	__SYSTEM.TYPE_CLASS.TYPE_STRING:
	
	convertResult := TryConvert_LINT_TO_STRING(in, _STRING);
	IF convertResult THEN
		convertAddress := ADR(_STRING);
	END_IF
	
END_CASE

IF convertResult THEN
	memcpy(out.pValue,convertAddress,DINT_TO_UDINT(out.diSize));
END_IF

TryConvert_LINT_TO_Destination := convertResult;

END_FUNCTION

// mobject-converters/Converters/LINT_TO_/TryConvert_LINT_TO_WORD
FUNCTION TryConvert_LINT_TO_WORD : BOOL
VAR_INPUT
	in : LINT;
	out : REFERENCE TO WORD;
END_VAR

IF in > DatatypeLimits.MAX_VALUE_OF_LINT_WHICH_CAN_BE_HELD_IN_A_WORD THEN
	RETURN;
END_IF

IF in < DatatypeLimits.MIN_VALUE_OF_LINT_WHICH_CAN_BE_HELD_IN_A_WORD THEN
	RETURN;
END_IF

out := LINT_TO_WORD(in);
TryConvert_LINT_TO_WORD := TRUE;

END_FUNCTION

// mobject-converters/Converters/LINT_TO_/TryConvert_LINT_TO_DWORD
FUNCTION TryConvert_LINT_TO_DWORD : BOOL
VAR_INPUT
	in : LINT;
	out : REFERENCE TO DWORD;
END_VAR

IF in > DatatypeLimits.MAX_VALUE_OF_LINT_WHICH_CAN_BE_HELD_IN_A_DWORD THEN
	RETURN;
END_IF

IF in < DatatypeLimits.MIN_VALUE_OF_LINT_WHICH_CAN_BE_HELD_IN_A_DWORD THEN
	RETURN;
END_IF

out := LINT_TO_DWORD(in);
TryConvert_LINT_TO_DWORD := TRUE;

END_FUNCTION

// mobject-converters/Converters/LINT_TO_/TryConvert_LINT_TO_LWORD
FUNCTION TryConvert_LINT_TO_LWORD : BOOL
VAR_INPUT
	in : LINT;
	out : REFERENCE TO LWORD;
END_VAR

IF in < DatatypeLimits.MIN_VALUE_OF_LINT_WHICH_CAN_BE_HELD_IN_A_LWORD THEN
	RETURN;
END_IF

out := LINT_TO_LWORD(in);
TryConvert_LINT_TO_LWORD := TRUE;

END_FUNCTION

// mobject-converters/Converters/LINT_TO_/TryConvert_LINT_TO_SINT
FUNCTION TryConvert_LINT_TO_SINT : BOOL
VAR_INPUT
	in : LINT;
	out : REFERENCE TO SINT;
END_VAR

IF in > DatatypeLimits.MAX_VALUE_OF_LINT_WHICH_CAN_BE_HELD_IN_A_SINT THEN
	RETURN;
END_IF

IF in < DatatypeLimits.MIN_VALUE_OF_LINT_WHICH_CAN_BE_HELD_IN_A_SINT THEN
	RETURN;
END_IF

out := LINT_TO_SINT(in);
TryConvert_LINT_TO_SINT := TRUE;

END_FUNCTION

// mobject-converters/Converters/LINT_TO_/TryConvert_LINT_TO_INT
FUNCTION TryConvert_LINT_TO_INT : BOOL
VAR_INPUT
	in : LINT;
	out : REFERENCE TO INT;
END_VAR

IF in > DatatypeLimits.MAX_VALUE_OF_LINT_WHICH_CAN_BE_HELD_IN_A_INT THEN
	RETURN;
END_IF

IF in < DatatypeLimits.MIN_VALUE_OF_LINT_WHICH_CAN_BE_HELD_IN_A_INT THEN
	RETURN;
END_IF

out := LINT_TO_INT(in);
TryConvert_LINT_TO_INT := TRUE;

END_FUNCTION

// mobject-converters/Converters/LINT_TO_/TryConvert_LINT_TO_DINT
FUNCTION TryConvert_LINT_TO_DINT : BOOL
VAR_INPUT
	in : LINT;
	out : REFERENCE TO DINT;
END_VAR

IF in > DatatypeLimits.MAX_VALUE_OF_LINT_WHICH_CAN_BE_HELD_IN_A_DINT THEN
	RETURN;
END_IF

IF in < DatatypeLimits.MIN_VALUE_OF_LINT_WHICH_CAN_BE_HELD_IN_A_DINT THEN
	RETURN;
END_IF

out := LINT_TO_DINT(in);
TryConvert_LINT_TO_DINT := TRUE;

END_FUNCTION

// mobject-converters/Converters/LINT_TO_/TryConvert_LINT_TO_LINT
FUNCTION TryConvert_LINT_TO_LINT : BOOL
VAR_INPUT
	in : LINT;
	out : REFERENCE TO LINT;
END_VAR

out := in;
TryConvert_LINT_TO_LINT := TRUE;

END_FUNCTION

// mobject-converters/Converters/LINT_TO_/TryConvert_LINT_TO_USINT
FUNCTION TryConvert_LINT_TO_USINT : BOOL
VAR_INPUT
	in : LINT;
	out : REFERENCE TO USINT;
END_VAR

IF in > DatatypeLimits.MAX_VALUE_OF_LINT_WHICH_CAN_BE_HELD_IN_A_USINT THEN
	RETURN;
END_IF

IF in < DatatypeLimits.MIN_VALUE_OF_LINT_WHICH_CAN_BE_HELD_IN_A_USINT THEN
	RETURN;
END_IF

out := LINT_TO_USINT(in);
TryConvert_LINT_TO_USINT := TRUE;

END_FUNCTION

// mobject-converters/Converters/LINT_TO_/TryConvert_LINT_TO_UINT
FUNCTION TryConvert_LINT_TO_UINT : BOOL
VAR_INPUT
	in : LINT;
	out : REFERENCE TO UINT;
END_VAR

IF in > DatatypeLimits.MAX_VALUE_OF_LINT_WHICH_CAN_BE_HELD_IN_A_UINT THEN
	RETURN;
END_IF

IF in < DatatypeLimits.MIN_VALUE_OF_LINT_WHICH_CAN_BE_HELD_IN_A_UINT THEN
	RETURN;
END_IF

out := LINT_TO_UINT(in);
TryConvert_LINT_TO_UINT := TRUE;

END_FUNCTION

// mobject-converters/Converters/LINT_TO_/TryConvert_LINT_TO_UDINT
FUNCTION TryConvert_LINT_TO_UDINT : BOOL
VAR_INPUT
	in : LINT;
	out : REFERENCE TO UDINT;
END_VAR

IF in > DatatypeLimits.MAX_VALUE_OF_LINT_WHICH_CAN_BE_HELD_IN_A_UDINT THEN
	RETURN;
END_IF

IF in < DatatypeLimits.MIN_VALUE_OF_LINT_WHICH_CAN_BE_HELD_IN_A_UDINT THEN
	RETURN;
END_IF

out := LINT_TO_UDINT(in);
TryConvert_LINT_TO_UDINT := TRUE;

END_FUNCTION

// mobject-converters/Converters/LINT_TO_/TryConvert_LINT_TO_ULINT
FUNCTION TryConvert_LINT_TO_ULINT : BOOL
VAR_INPUT
	in : LINT;
	out : REFERENCE TO ULINT;
END_VAR

IF in < DatatypeLimits.MIN_VALUE_OF_LINT_WHICH_CAN_BE_HELD_IN_A_ULINT THEN
	RETURN;
END_IF

out := LINT_TO_ULINT(in);
TryConvert_LINT_TO_ULINT := TRUE;

END_FUNCTION

// mobject-converters/Converters/LINT_TO_/TryConvert_LINT_TO_REAL
FUNCTION TryConvert_LINT_TO_REAL : BOOL
VAR_INPUT
	in : LINT;
	out : REFERENCE TO REAL;
END_VAR

out := LINT_TO_REAL(in);
TryConvert_LINT_TO_REAL := TRUE;

END_FUNCTION

// mobject-converters/Converters/LINT_TO_/TryConvert_LINT_TO_LREAL
FUNCTION TryConvert_LINT_TO_LREAL : BOOL
VAR_INPUT
	in : LINT;
	out : REFERENCE TO LREAL;
END_VAR

out := LINT_TO_LREAL(in);
TryConvert_LINT_TO_LREAL := TRUE;

END_FUNCTION

// mobject-converters/Converters/LINT_TO_/TryConvert_LINT_TO_TIME
FUNCTION TryConvert_LINT_TO_TIME : BOOL
VAR_INPUT
	in : LINT;
	out : REFERENCE TO TIME;
END_VAR

IF in > DatatypeLimits.MAX_VALUE_OF_LINT_WHICH_CAN_BE_HELD_IN_A_TIME THEN
	RETURN;
END_IF

IF in < DatatypeLimits.MIN_VALUE_OF_LINT_WHICH_CAN_BE_HELD_IN_A_TIME THEN
	RETURN;
END_IF

out := LINT_TO_TIME(in);
TryConvert_LINT_TO_TIME := TRUE;

END_FUNCTION

// mobject-converters/Converters/LINT_TO_/TryConvert_LINT_TO_TOD
FUNCTION TryConvert_LINT_TO_TOD : BOOL
VAR_INPUT
	in : LINT;
	out : REFERENCE TO TOD;
END_VAR

IF in > DatatypeLimits.MAX_VALUE_OF_LINT_WHICH_CAN_BE_HELD_IN_A_TOD THEN
	RETURN;
END_IF

IF in < DatatypeLimits.MIN_VALUE_OF_LINT_WHICH_CAN_BE_HELD_IN_A_TOD THEN
	RETURN;
END_IF

out := LINT_TO_TOD(in);
TryConvert_LINT_TO_TOD := TRUE;

END_FUNCTION

// mobject-converters/Converters/LINT_TO_/TryConvert_LINT_TO_DT
FUNCTION TryConvert_LINT_TO_DT : BOOL
VAR_INPUT
	in : LINT;
	out : REFERENCE TO DT;
END_VAR

IF in > DatatypeLimits.MAX_VALUE_OF_LINT_WHICH_CAN_BE_HELD_IN_A_DT THEN
	RETURN;
END_IF

IF in < DatatypeLimits.MIN_VALUE_OF_LINT_WHICH_CAN_BE_HELD_IN_A_DT THEN
	RETURN;
END_IF

out := LINT_TO_DT(in);
TryConvert_LINT_TO_DT := TRUE;

END_FUNCTION

// mobject-converters/Converters/LINT_TO_/TryConvert_LINT_TO_STRING
FUNCTION TryConvert_LINT_TO_STRING : BOOL
VAR_INPUT
	in : LINT;
	out : REFERENCE TO STRING;
END_VAR

out := LINT_TO_STRING(in);
TryConvert_LINT_TO_STRING := TRUE;

END_FUNCTION

// mobject-converters/Converters/LREAL_TO_/TryConvert_LREAL_TO_BOOL
FUNCTION TryConvert_LREAL_TO_BOOL : BOOL
VAR_INPUT
	in : LREAL;
	out : REFERENCE TO BOOL;
END_VAR

out := LREAL_TO_BOOL(in);
TryConvert_LREAL_TO_BOOL := TRUE;

END_FUNCTION

// mobject-converters/Converters/LREAL_TO_/TryConvert_LREAL_TO_BYTE
FUNCTION TryConvert_LREAL_TO_BYTE : BOOL
VAR_INPUT
	in : LREAL;
	out : REFERENCE TO BYTE;
END_VAR

IF in > DatatypeLimits.MAX_VALUE_OF_LREAL_WHICH_CAN_BE_HELD_IN_A_BYTE THEN
	RETURN;
END_IF

IF in < DatatypeLimits.MIN_VALUE_OF_LREAL_WHICH_CAN_BE_HELD_IN_A_BYTE THEN
	RETURN;
END_IF

out := LREAL_TO_BYTE(in);
TryConvert_LREAL_TO_BYTE := TRUE;

END_FUNCTION

// mobject-converters/Converters/LREAL_TO_/TryConvert_LREAL_TO_DATE
FUNCTION TryConvert_LREAL_TO_DATE : BOOL
VAR_INPUT
	in : LREAL;
	out : REFERENCE TO DATE;
END_VAR

IF in > DatatypeLimits.MAX_VALUE_OF_LREAL_WHICH_CAN_BE_HELD_IN_A_DATE THEN
	RETURN;
END_IF

IF in < DatatypeLimits.MIN_VALUE_OF_LREAL_WHICH_CAN_BE_HELD_IN_A_DATE THEN
	RETURN;
END_IF

out := LREAL_TO_DATE(in);
TryConvert_LREAL_TO_DATE := TRUE;

END_FUNCTION

// mobject-converters/Converters/LREAL_TO_/TryConvert_LREAL_TO_Destination
FUNCTION TryConvert_LREAL_TO_Destination : BOOL
VAR_INPUT
	in : LREAL;
	out : ANY;
END_VAR
VAR
	convertResult : BOOL := FALSE;
	convertAddress : PVOID;
	_BOOL : BOOL;
	_BYTE : BYTE;
	_WORD : WORD;
	_DWORD : DWORD;
	_LWORD : LWORD;
	_SINT : SINT;
	_INT : INT;
	_DINT : DINT;
	_LINT : LINT;
	_USINT : USINT;
	_UINT : UINT;
	_UDINT : UDINT;
	_ULINT : ULINT;
	_REAL : REAL;
	_LREAL : LREAL;
	_TIME : TIME;
	_TOD : TOD;
	_DATE : DATE;
	_DT : DT;
	_STRING : STRING;
END_VAR

CASE out.TypeClass OF
	__SYSTEM.TYPE_CLASS.TYPE_BOOL:
	
	convertResult := TryConvert_LREAL_TO_BOOL(in, _BOOL);
	IF convertResult THEN
		convertAddress := ADR(_BOOL);
	END_IF
	
	__SYSTEM.TYPE_CLASS.TYPE_BYTE:
	
	convertResult := TryConvert_LREAL_TO_BYTE(in, _BYTE);
	IF convertResult THEN
		convertAddress := ADR(_BYTE);
	END_IF
	
	__SYSTEM.TYPE_CLASS.TYPE_WORD:
	
	convertResult := TryConvert_LREAL_TO_WORD(in, _WORD);
	IF convertResult THEN
		convertAddress := ADR(_WORD);
	END_IF
	
	__SYSTEM.TYPE_CLASS.TYPE_DWORD:
	
	convertResult := TryConvert_LREAL_TO_DWORD(in, _DWORD);
	IF convertResult THEN
		convertAddress := ADR(_DWORD);
	END_IF
	
	__SYSTEM.TYPE_CLASS.TYPE_LWORD:
	
	convertResult := TryConvert_LREAL_TO_LWORD(in, _LWORD);
	IF convertResult THEN
		convertAddress := ADR(_LWORD);
	END_IF
	
	__SYSTEM.TYPE_CLASS.TYPE_SINT:
	
	convertResult := TryConvert_LREAL_TO_SINT(in, _SINT);
	IF convertResult THEN
		convertAddress := ADR(_SINT);
	END_IF
	
	__SYSTEM.TYPE_CLASS.TYPE_INT:
	
	convertResult := TryConvert_LREAL_TO_INT(in, _INT);
	IF convertResult THEN
		convertAddress := ADR(_INT);
	END_IF
	
	__SYSTEM.TYPE_CLASS.TYPE_DINT:
	
	convertResult := TryConvert_LREAL_TO_DINT(in, _DINT);
	IF convertResult THEN
		convertAddress := ADR(_DINT);
	END_IF
	
	__SYSTEM.TYPE_CLASS.TYPE_LINT:
	
	convertResult := TryConvert_LREAL_TO_LINT(in, _LINT);
	IF convertResult THEN
		convertAddress := ADR(_LINT);
	END_IF
	
	__SYSTEM.TYPE_CLASS.TYPE_USINT:
	
	convertResult := TryConvert_LREAL_TO_USINT(in, _USINT);
	IF convertResult THEN
		convertAddress := ADR(_USINT);
	END_IF
	
	__SYSTEM.TYPE_CLASS.TYPE_UINT:
	
	convertResult := TryConvert_LREAL_TO_UINT(in, _UINT);
	IF convertResult THEN
		convertAddress := ADR(_UINT);
	END_IF
	
	__SYSTEM.TYPE_CLASS.TYPE_UDINT:
	
	convertResult := TryConvert_LREAL_TO_UDINT(in, _UDINT);
	IF convertResult THEN
		convertAddress := ADR(_UDINT);
	END_IF
	
	__SYSTEM.TYPE_CLASS.TYPE_ULINT:
	
	convertResult := TryConvert_LREAL_TO_ULINT(in, _ULINT);
	IF convertResult THEN
		convertAddress := ADR(_ULINT);
	END_IF
	
	__SYSTEM.TYPE_CLASS.TYPE_REAL:
	
	convertResult := TryConvert_LREAL_TO_REAL(in, _REAL);
	IF convertResult THEN
		convertAddress := ADR(_REAL);
	END_IF
	
	__SYSTEM.TYPE_CLASS.TYPE_LREAL:
	
	convertResult := TryConvert_LREAL_TO_LREAL(in, _LREAL);
	IF convertResult THEN
		convertAddress := ADR(_LREAL);
	END_IF
	
	__SYSTEM.TYPE_CLASS.TYPE_TIME:
	
	convertResult := TryConvert_LREAL_TO_TIME(in, _TIME);
	IF convertResult THEN
		convertAddress := ADR(_TIME);
	END_IF
	
	__SYSTEM.TYPE_CLASS.TYPE_TIMEOFDAY:
	
	convertResult := TryConvert_LREAL_TO_TOD(in, _TOD);
	IF convertResult THEN
		convertAddress := ADR(_TOD);
	END_IF
	
	__SYSTEM.TYPE_CLASS.TYPE_DATE:
	
	convertResult := TryConvert_LREAL_TO_DATE(in, _DATE);
	IF convertResult THEN
		convertAddress := ADR(_DATE);
	END_IF
	
	__SYSTEM.TYPE_CLASS.TYPE_DATEANDTIME:
	
	convertResult := TryConvert_LREAL_TO_DT(in, _DT);
	IF convertResult THEN
		convertAddress := ADR(_DT);
	END_IF
	
	__SYSTEM.TYPE_CLASS.TYPE_STRING:
	
	convertResult := TryConvert_LREAL_TO_STRING(in, _STRING);
	IF convertResult THEN
		convertAddress := ADR(_STRING);
	END_IF
	
END_CASE

IF convertResult THEN
	memcpy(out.pValue,convertAddress,DINT_TO_UDINT(out.diSize));
END_IF

TryConvert_LREAL_TO_Destination := convertResult;

END_FUNCTION

// mobject-converters/Converters/LREAL_TO_/TryConvert_LREAL_TO_WORD
FUNCTION TryConvert_LREAL_TO_WORD : BOOL
VAR_INPUT
	in : LREAL;
	out : REFERENCE TO WORD;
END_VAR

IF in > DatatypeLimits.MAX_VALUE_OF_LREAL_WHICH_CAN_BE_HELD_IN_A_WORD THEN
	RETURN;
END_IF

IF in < DatatypeLimits.MIN_VALUE_OF_LREAL_WHICH_CAN_BE_HELD_IN_A_WORD THEN
	RETURN;
END_IF

out := LREAL_TO_WORD(in);
TryConvert_LREAL_TO_WORD := TRUE;

END_FUNCTION

// mobject-converters/Converters/LREAL_TO_/TryConvert_LREAL_TO_DWORD
FUNCTION TryConvert_LREAL_TO_DWORD : BOOL
VAR_INPUT
	in : LREAL;
	out : REFERENCE TO DWORD;
END_VAR

IF in > DatatypeLimits.MAX_VALUE_OF_LREAL_WHICH_CAN_BE_HELD_IN_A_DWORD THEN
	RETURN;
END_IF

IF in < DatatypeLimits.MIN_VALUE_OF_LREAL_WHICH_CAN_BE_HELD_IN_A_DWORD THEN
	RETURN;
END_IF

out := LREAL_TO_DWORD(in);
TryConvert_LREAL_TO_DWORD := TRUE;

END_FUNCTION

// mobject-converters/Converters/LREAL_TO_/TryConvert_LREAL_TO_LWORD
FUNCTION TryConvert_LREAL_TO_LWORD : BOOL
VAR_INPUT
	in : LREAL;
	out : REFERENCE TO LWORD;
END_VAR

IF in > DatatypeLimits.MAX_VALUE_OF_LREAL_WHICH_CAN_BE_HELD_IN_A_LWORD THEN
	RETURN;
END_IF

IF in < DatatypeLimits.MIN_VALUE_OF_LREAL_WHICH_CAN_BE_HELD_IN_A_LWORD THEN
	RETURN;
END_IF

out := LREAL_TO_LWORD(in);
TryConvert_LREAL_TO_LWORD := TRUE;

END_FUNCTION

// mobject-converters/Converters/LREAL_TO_/TryConvert_LREAL_TO_SINT
FUNCTION TryConvert_LREAL_TO_SINT : BOOL
VAR_INPUT
	in : LREAL;
	out : REFERENCE TO SINT;
END_VAR

IF in > DatatypeLimits.MAX_VALUE_OF_LREAL_WHICH_CAN_BE_HELD_IN_A_SINT THEN
	RETURN;
END_IF

IF in < DatatypeLimits.MIN_VALUE_OF_LREAL_WHICH_CAN_BE_HELD_IN_A_SINT THEN
	RETURN;
END_IF

out := LREAL_TO_SINT(in);
TryConvert_LREAL_TO_SINT := TRUE;

END_FUNCTION

// mobject-converters/Converters/LREAL_TO_/TryConvert_LREAL_TO_INT
FUNCTION TryConvert_LREAL_TO_INT : BOOL
VAR_INPUT
	in : LREAL;
	out : REFERENCE TO INT;
END_VAR

IF in > DatatypeLimits.MAX_VALUE_OF_LREAL_WHICH_CAN_BE_HELD_IN_A_INT THEN
	RETURN;
END_IF

IF in < DatatypeLimits.MIN_VALUE_OF_LREAL_WHICH_CAN_BE_HELD_IN_A_INT THEN
	RETURN;
END_IF

out := LREAL_TO_INT(in);
TryConvert_LREAL_TO_INT := TRUE;

END_FUNCTION

// mobject-converters/Converters/LREAL_TO_/TryConvert_LREAL_TO_DINT
FUNCTION TryConvert_LREAL_TO_DINT : BOOL
VAR_INPUT
	in : LREAL;
	out : REFERENCE TO DINT;
END_VAR

IF in > DatatypeLimits.MAX_VALUE_OF_LREAL_WHICH_CAN_BE_HELD_IN_A_DINT THEN
	RETURN;
END_IF

IF in < DatatypeLimits.MIN_VALUE_OF_LREAL_WHICH_CAN_BE_HELD_IN_A_DINT THEN
	RETURN;
END_IF

out := LREAL_TO_DINT(in);
TryConvert_LREAL_TO_DINT := TRUE;

END_FUNCTION

// mobject-converters/Converters/LREAL_TO_/TryConvert_LREAL_TO_LINT
FUNCTION TryConvert_LREAL_TO_LINT : BOOL
VAR_INPUT
	in : LREAL;
	out : REFERENCE TO LINT;
END_VAR

IF in > DatatypeLimits.MAX_VALUE_OF_LREAL_WHICH_CAN_BE_HELD_IN_A_LINT THEN
	RETURN;
END_IF

IF in < DatatypeLimits.MIN_VALUE_OF_LREAL_WHICH_CAN_BE_HELD_IN_A_LINT THEN
	RETURN;
END_IF

out := LREAL_TO_LINT(in);
TryConvert_LREAL_TO_LINT := TRUE;

END_FUNCTION

// mobject-converters/Converters/LREAL_TO_/TryConvert_LREAL_TO_USINT
FUNCTION TryConvert_LREAL_TO_USINT : BOOL
VAR_INPUT
	in : LREAL;
	out : REFERENCE TO USINT;
END_VAR

IF in > DatatypeLimits.MAX_VALUE_OF_LREAL_WHICH_CAN_BE_HELD_IN_A_USINT THEN
	RETURN;
END_IF

IF in < DatatypeLimits.MIN_VALUE_OF_LREAL_WHICH_CAN_BE_HELD_IN_A_USINT THEN
	RETURN;
END_IF

out := LREAL_TO_USINT(in);
TryConvert_LREAL_TO_USINT := TRUE;

END_FUNCTION

// mobject-converters/Converters/LREAL_TO_/TryConvert_LREAL_TO_UINT
FUNCTION TryConvert_LREAL_TO_UINT : BOOL
VAR_INPUT
	in : LREAL;
	out : REFERENCE TO UINT;
END_VAR

IF in > DatatypeLimits.MAX_VALUE_OF_LREAL_WHICH_CAN_BE_HELD_IN_A_UINT THEN
	RETURN;
END_IF

IF in < DatatypeLimits.MIN_VALUE_OF_LREAL_WHICH_CAN_BE_HELD_IN_A_UINT THEN
	RETURN;
END_IF

out := LREAL_TO_UINT(in);
TryConvert_LREAL_TO_UINT := TRUE;

END_FUNCTION

// mobject-converters/Converters/LREAL_TO_/TryConvert_LREAL_TO_UDINT
FUNCTION TryConvert_LREAL_TO_UDINT : BOOL
VAR_INPUT
	in : LREAL;
	out : REFERENCE TO UDINT;
END_VAR

IF in > DatatypeLimits.MAX_VALUE_OF_LREAL_WHICH_CAN_BE_HELD_IN_A_UDINT THEN
	RETURN;
END_IF

IF in < DatatypeLimits.MIN_VALUE_OF_LREAL_WHICH_CAN_BE_HELD_IN_A_UDINT THEN
	RETURN;
END_IF

out := LREAL_TO_UDINT(in);
TryConvert_LREAL_TO_UDINT := TRUE;

END_FUNCTION

// mobject-converters/Converters/LREAL_TO_/TryConvert_LREAL_TO_ULINT
FUNCTION TryConvert_LREAL_TO_ULINT : BOOL
VAR_INPUT
	in : LREAL;
	out : REFERENCE TO ULINT;
END_VAR

IF in > DatatypeLimits.MAX_VALUE_OF_LREAL_WHICH_CAN_BE_HELD_IN_A_ULINT THEN
	RETURN;
END_IF

IF in < DatatypeLimits.MIN_VALUE_OF_LREAL_WHICH_CAN_BE_HELD_IN_A_ULINT THEN
	RETURN;
END_IF

out := LREAL_TO_ULINT(in);
TryConvert_LREAL_TO_ULINT := TRUE;

END_FUNCTION

// mobject-converters/Converters/LREAL_TO_/TryConvert_LREAL_TO_REAL
FUNCTION TryConvert_LREAL_TO_REAL : BOOL
VAR_INPUT
	in : LREAL;
	out : REFERENCE TO REAL;
END_VAR

IF in > DatatypeLimits.MAX_VALUE_OF_LREAL_WHICH_CAN_BE_HELD_IN_A_REAL THEN
	RETURN;
END_IF

IF in < DatatypeLimits.MIN_VALUE_OF_LREAL_WHICH_CAN_BE_HELD_IN_A_REAL THEN
	RETURN;
END_IF

out := LREAL_TO_REAL(in);
TryConvert_LREAL_TO_REAL := TRUE;

END_FUNCTION

// mobject-converters/Converters/LREAL_TO_/TryConvert_LREAL_TO_LREAL
FUNCTION TryConvert_LREAL_TO_LREAL : BOOL
VAR_INPUT
	in : LREAL;
	out : REFERENCE TO LREAL;
END_VAR

out := in;
TryConvert_LREAL_TO_LREAL := TRUE;

END_FUNCTION

// mobject-converters/Converters/LREAL_TO_/TryConvert_LREAL_TO_TIME
FUNCTION TryConvert_LREAL_TO_TIME : BOOL
VAR_INPUT
	in : LREAL;
	out : REFERENCE TO TIME;
END_VAR

IF in > DatatypeLimits.MAX_VALUE_OF_LREAL_WHICH_CAN_BE_HELD_IN_A_TIME THEN
	RETURN;
END_IF

IF in < DatatypeLimits.MIN_VALUE_OF_LREAL_WHICH_CAN_BE_HELD_IN_A_TIME THEN
	RETURN;
END_IF

out := LREAL_TO_TIME(in);
TryConvert_LREAL_TO_TIME := TRUE;

END_FUNCTION

// mobject-converters/Converters/LREAL_TO_/TryConvert_LREAL_TO_TOD
FUNCTION TryConvert_LREAL_TO_TOD : BOOL
VAR_INPUT
	in : LREAL;
	out : REFERENCE TO TOD;
END_VAR

IF in > DatatypeLimits.MAX_VALUE_OF_LREAL_WHICH_CAN_BE_HELD_IN_A_TOD THEN
	RETURN;
END_IF

IF in < DatatypeLimits.MIN_VALUE_OF_LREAL_WHICH_CAN_BE_HELD_IN_A_TOD THEN
	RETURN;
END_IF

out := LREAL_TO_TOD(in);
TryConvert_LREAL_TO_TOD := TRUE;

END_FUNCTION

// mobject-converters/Converters/LREAL_TO_/TryConvert_LREAL_TO_DT
FUNCTION TryConvert_LREAL_TO_DT : BOOL
VAR_INPUT
	in : LREAL;
	out : REFERENCE TO DT;
END_VAR

IF in > DatatypeLimits.MAX_VALUE_OF_LREAL_WHICH_CAN_BE_HELD_IN_A_DT THEN
	RETURN;
END_IF

IF in < DatatypeLimits.MIN_VALUE_OF_LREAL_WHICH_CAN_BE_HELD_IN_A_DT THEN
	RETURN;
END_IF

out := LREAL_TO_DT(in);
TryConvert_LREAL_TO_DT := TRUE;

END_FUNCTION

// mobject-converters/Converters/LREAL_TO_/TryConvert_LREAL_TO_STRING
FUNCTION TryConvert_LREAL_TO_STRING : BOOL
VAR_INPUT
	in : LREAL;
	out : REFERENCE TO STRING;
END_VAR

IF in > DatatypeLimits.MAX_VALUE_OF_LREAL_WHICH_CAN_BE_HELD_IN_A_STRING THEN
	RETURN;
END_IF

IF in < DatatypeLimits.MIN_VALUE_OF_LREAL_WHICH_CAN_BE_HELD_IN_A_STRING THEN
	RETURN;
END_IF

out := LREAL_TO_STRING(in);
TryConvert_LREAL_TO_STRING := TRUE;

END_FUNCTION

// mobject-converters/Converters/LWORD_TO_/TryConvert_LWORD_TO_BOOL
FUNCTION TryConvert_LWORD_TO_BOOL : BOOL
VAR_INPUT
	in : LWORD;
	out : REFERENCE TO BOOL;
END_VAR

out := LWORD_TO_BOOL(in);
TryConvert_LWORD_TO_BOOL := TRUE;

END_FUNCTION

// mobject-converters/Converters/LWORD_TO_/TryConvert_LWORD_TO_BYTE
FUNCTION TryConvert_LWORD_TO_BYTE : BOOL
VAR_INPUT
	in : LWORD;
	out : REFERENCE TO BYTE;
END_VAR

IF in > DatatypeLimits.MAX_VALUE_OF_LWORD_WHICH_CAN_BE_HELD_IN_A_BYTE THEN
	RETURN;
END_IF

out := LWORD_TO_BYTE(in);
TryConvert_LWORD_TO_BYTE := TRUE;

END_FUNCTION

// mobject-converters/Converters/LWORD_TO_/TryConvert_LWORD_TO_DATE
FUNCTION TryConvert_LWORD_TO_DATE : BOOL
VAR_INPUT
	in : LWORD;
	out : REFERENCE TO DATE;
END_VAR

IF in > DatatypeLimits.MAX_VALUE_OF_LWORD_WHICH_CAN_BE_HELD_IN_A_DATE THEN
	RETURN;
END_IF

out := LWORD_TO_DATE(in);
TryConvert_LWORD_TO_DATE := TRUE;

END_FUNCTION

// mobject-converters/Converters/LWORD_TO_/TryConvert_LWORD_TO_Destination
FUNCTION TryConvert_LWORD_TO_Destination : BOOL
VAR_INPUT
	in : LWORD;
	out : ANY;
END_VAR
VAR
	convertResult : BOOL := FALSE;
	convertAddress : PVOID;
	_BOOL : BOOL;
	_BYTE : BYTE;
	_WORD : WORD;
	_DWORD : DWORD;
	_LWORD : LWORD;
	_SINT : SINT;
	_INT : INT;
	_DINT : DINT;
	_LINT : LINT;
	_USINT : USINT;
	_UINT : UINT;
	_UDINT : UDINT;
	_ULINT : ULINT;
	_REAL : REAL;
	_LREAL : LREAL;
	_TIME : TIME;
	_TOD : TOD;
	_DATE : DATE;
	_DT : DT;
	_STRING : STRING;
END_VAR

CASE out.TypeClass OF
	__SYSTEM.TYPE_CLASS.TYPE_BOOL:
	
	convertResult := TryConvert_LWORD_TO_BOOL(in, _BOOL);
	IF convertResult THEN
		convertAddress := ADR(_BOOL);
	END_IF
	
	__SYSTEM.TYPE_CLASS.TYPE_BYTE:
	
	convertResult := TryConvert_LWORD_TO_BYTE(in, _BYTE);
	IF convertResult THEN
		convertAddress := ADR(_BYTE);
	END_IF
	
	__SYSTEM.TYPE_CLASS.TYPE_WORD:
	
	convertResult := TryConvert_LWORD_TO_WORD(in, _WORD);
	IF convertResult THEN
		convertAddress := ADR(_WORD);
	END_IF
	
	__SYSTEM.TYPE_CLASS.TYPE_DWORD:
	
	convertResult := TryConvert_LWORD_TO_DWORD(in, _DWORD);
	IF convertResult THEN
		convertAddress := ADR(_DWORD);
	END_IF
	
	__SYSTEM.TYPE_CLASS.TYPE_LWORD:
	
	convertResult := TryConvert_LWORD_TO_LWORD(in, _LWORD);
	IF convertResult THEN
		convertAddress := ADR(_LWORD);
	END_IF
	
	__SYSTEM.TYPE_CLASS.TYPE_SINT:
	
	convertResult := TryConvert_LWORD_TO_SINT(in, _SINT);
	IF convertResult THEN
		convertAddress := ADR(_SINT);
	END_IF
	
	__SYSTEM.TYPE_CLASS.TYPE_INT:
	
	convertResult := TryConvert_LWORD_TO_INT(in, _INT);
	IF convertResult THEN
		convertAddress := ADR(_INT);
	END_IF
	
	__SYSTEM.TYPE_CLASS.TYPE_DINT:
	
	convertResult := TryConvert_LWORD_TO_DINT(in, _DINT);
	IF convertResult THEN
		convertAddress := ADR(_DINT);
	END_IF
	
	__SYSTEM.TYPE_CLASS.TYPE_LINT:
	
	convertResult := TryConvert_LWORD_TO_LINT(in, _LINT);
	IF convertResult THEN
		convertAddress := ADR(_LINT);
	END_IF
	
	__SYSTEM.TYPE_CLASS.TYPE_USINT:
	
	convertResult := TryConvert_LWORD_TO_USINT(in, _USINT);
	IF convertResult THEN
		convertAddress := ADR(_USINT);
	END_IF
	
	__SYSTEM.TYPE_CLASS.TYPE_UINT:
	
	convertResult := TryConvert_LWORD_TO_UINT(in, _UINT);
	IF convertResult THEN
		convertAddress := ADR(_UINT);
	END_IF
	
	__SYSTEM.TYPE_CLASS.TYPE_UDINT:
	
	convertResult := TryConvert_LWORD_TO_UDINT(in, _UDINT);
	IF convertResult THEN
		convertAddress := ADR(_UDINT);
	END_IF
	
	__SYSTEM.TYPE_CLASS.TYPE_ULINT:
	
	convertResult := TryConvert_LWORD_TO_ULINT(in, _ULINT);
	IF convertResult THEN
		convertAddress := ADR(_ULINT);
	END_IF
	
	__SYSTEM.TYPE_CLASS.TYPE_REAL:
	
	convertResult := TryConvert_LWORD_TO_REAL(in, _REAL);
	IF convertResult THEN
		convertAddress := ADR(_REAL);
	END_IF
	
	__SYSTEM.TYPE_CLASS.TYPE_LREAL:
	
	convertResult := TryConvert_LWORD_TO_LREAL(in, _LREAL);
	IF convertResult THEN
		convertAddress := ADR(_LREAL);
	END_IF
	
	__SYSTEM.TYPE_CLASS.TYPE_TIME:
	
	convertResult := TryConvert_LWORD_TO_TIME(in, _TIME);
	IF convertResult THEN
		convertAddress := ADR(_TIME);
	END_IF
	
	__SYSTEM.TYPE_CLASS.TYPE_TIMEOFDAY:
	
	convertResult := TryConvert_LWORD_TO_TOD(in, _TOD);
	IF convertResult THEN
		convertAddress := ADR(_TOD);
	END_IF
	
	__SYSTEM.TYPE_CLASS.TYPE_DATE:
	
	convertResult := TryConvert_LWORD_TO_DATE(in, _DATE);
	IF convertResult THEN
		convertAddress := ADR(_DATE);
	END_IF
	
	__SYSTEM.TYPE_CLASS.TYPE_DATEANDTIME:
	
	convertResult := TryConvert_LWORD_TO_DT(in, _DT);
	IF convertResult THEN
		convertAddress := ADR(_DT);
	END_IF
	
	__SYSTEM.TYPE_CLASS.TYPE_STRING:
	
	convertResult := TryConvert_LWORD_TO_STRING(in, _STRING);
	IF convertResult THEN
		convertAddress := ADR(_STRING);
	END_IF
	
END_CASE

IF convertResult THEN
	memcpy(out.pValue,convertAddress,DINT_TO_UDINT(out.diSize));
END_IF

TryConvert_LWORD_TO_Destination := convertResult;

END_FUNCTION

// mobject-converters/Converters/LWORD_TO_/TryConvert_LWORD_TO_WORD
FUNCTION TryConvert_LWORD_TO_WORD : BOOL
VAR_INPUT
	in : LWORD;
	out : REFERENCE TO WORD;
END_VAR

IF in > DatatypeLimits.MAX_VALUE_OF_LWORD_WHICH_CAN_BE_HELD_IN_A_WORD THEN
	RETURN;
END_IF

out := LWORD_TO_WORD(in);
TryConvert_LWORD_TO_WORD := TRUE;

END_FUNCTION

// mobject-converters/Converters/LWORD_TO_/TryConvert_LWORD_TO_DWORD
FUNCTION TryConvert_LWORD_TO_DWORD : BOOL
VAR_INPUT
	in : LWORD;
	out : REFERENCE TO DWORD;
END_VAR

IF in > DatatypeLimits.MAX_VALUE_OF_LWORD_WHICH_CAN_BE_HELD_IN_A_DWORD THEN
	RETURN;
END_IF

out := LWORD_TO_DWORD(in);
TryConvert_LWORD_TO_DWORD := TRUE;

END_FUNCTION

// mobject-converters/Converters/LWORD_TO_/TryConvert_LWORD_TO_LWORD
FUNCTION TryConvert_LWORD_TO_LWORD : BOOL
VAR_INPUT
	in : LWORD;
	out : REFERENCE TO LWORD;
END_VAR

out := in;
TryConvert_LWORD_TO_LWORD := TRUE;

END_FUNCTION

// mobject-converters/Converters/LWORD_TO_/TryConvert_LWORD_TO_SINT
FUNCTION TryConvert_LWORD_TO_SINT : BOOL
VAR_INPUT
	in : LWORD;
	out : REFERENCE TO SINT;
END_VAR

IF in > DatatypeLimits.MAX_VALUE_OF_LWORD_WHICH_CAN_BE_HELD_IN_A_SINT THEN
	RETURN;
END_IF

out := LWORD_TO_SINT(in);
TryConvert_LWORD_TO_SINT := TRUE;

END_FUNCTION

// mobject-converters/Converters/LWORD_TO_/TryConvert_LWORD_TO_INT
FUNCTION TryConvert_LWORD_TO_INT : BOOL
VAR_INPUT
	in : LWORD;
	out : REFERENCE TO INT;
END_VAR

IF in > DatatypeLimits.MAX_VALUE_OF_LWORD_WHICH_CAN_BE_HELD_IN_A_INT THEN
	RETURN;
END_IF

out := LWORD_TO_INT(in);
TryConvert_LWORD_TO_INT := TRUE;

END_FUNCTION

// mobject-converters/Converters/LWORD_TO_/TryConvert_LWORD_TO_DINT
FUNCTION TryConvert_LWORD_TO_DINT : BOOL
VAR_INPUT
	in : LWORD;
	out : REFERENCE TO DINT;
END_VAR

IF in > DatatypeLimits.MAX_VALUE_OF_LWORD_WHICH_CAN_BE_HELD_IN_A_DINT THEN
	RETURN;
END_IF

out := LWORD_TO_DINT(in);
TryConvert_LWORD_TO_DINT := TRUE;

END_FUNCTION

// mobject-converters/Converters/LWORD_TO_/TryConvert_LWORD_TO_LINT
FUNCTION TryConvert_LWORD_TO_LINT : BOOL
VAR_INPUT
	in : LWORD;
	out : REFERENCE TO LINT;
END_VAR

IF in > DatatypeLimits.MAX_VALUE_OF_LWORD_WHICH_CAN_BE_HELD_IN_A_LINT THEN
	RETURN;
END_IF

out := LWORD_TO_LINT(in);
TryConvert_LWORD_TO_LINT := TRUE;

END_FUNCTION

// mobject-converters/Converters/LWORD_TO_/TryConvert_LWORD_TO_USINT
FUNCTION TryConvert_LWORD_TO_USINT : BOOL
VAR_INPUT
	in : LWORD;
	out : REFERENCE TO USINT;
END_VAR

IF in > DatatypeLimits.MAX_VALUE_OF_LWORD_WHICH_CAN_BE_HELD_IN_A_USINT THEN
	RETURN;
END_IF

out := LWORD_TO_USINT(in);
TryConvert_LWORD_TO_USINT := TRUE;

END_FUNCTION

// mobject-converters/Converters/LWORD_TO_/TryConvert_LWORD_TO_UINT
FUNCTION TryConvert_LWORD_TO_UINT : BOOL
VAR_INPUT
	in : LWORD;
	out : REFERENCE TO UINT;
END_VAR

IF in > DatatypeLimits.MAX_VALUE_OF_LWORD_WHICH_CAN_BE_HELD_IN_A_UINT THEN
	RETURN;
END_IF

out := LWORD_TO_UINT(in);
TryConvert_LWORD_TO_UINT := TRUE;

END_FUNCTION

// mobject-converters/Converters/LWORD_TO_/TryConvert_LWORD_TO_UDINT
FUNCTION TryConvert_LWORD_TO_UDINT : BOOL
VAR_INPUT
	in : LWORD;
	out : REFERENCE TO UDINT;
END_VAR

IF in > DatatypeLimits.MAX_VALUE_OF_LWORD_WHICH_CAN_BE_HELD_IN_A_UDINT THEN
	RETURN;
END_IF

out := LWORD_TO_UDINT(in);
TryConvert_LWORD_TO_UDINT := TRUE;

END_FUNCTION

// mobject-converters/Converters/LWORD_TO_/TryConvert_LWORD_TO_ULINT
FUNCTION TryConvert_LWORD_TO_ULINT : BOOL
VAR_INPUT
	in : LWORD;
	out : REFERENCE TO ULINT;
END_VAR

out := LWORD_TO_ULINT(in);
TryConvert_LWORD_TO_ULINT := TRUE;

END_FUNCTION

// mobject-converters/Converters/LWORD_TO_/TryConvert_LWORD_TO_REAL
FUNCTION TryConvert_LWORD_TO_REAL : BOOL
VAR_INPUT
	in : LWORD;
	out : REFERENCE TO REAL;
END_VAR

out := LWORD_TO_REAL(in);
TryConvert_LWORD_TO_REAL := TRUE;

END_FUNCTION

// mobject-converters/Converters/LWORD_TO_/TryConvert_LWORD_TO_LREAL
FUNCTION TryConvert_LWORD_TO_LREAL : BOOL
VAR_INPUT
	in : LWORD;
	out : REFERENCE TO LREAL;
END_VAR

out := LWORD_TO_LREAL(in);
TryConvert_LWORD_TO_LREAL := TRUE;

END_FUNCTION

// mobject-converters/Converters/LWORD_TO_/TryConvert_LWORD_TO_TIME
FUNCTION TryConvert_LWORD_TO_TIME : BOOL
VAR_INPUT
	in : LWORD;
	out : REFERENCE TO TIME;
END_VAR

IF in > DatatypeLimits.MAX_VALUE_OF_LWORD_WHICH_CAN_BE_HELD_IN_A_TIME THEN
	RETURN;
END_IF

out := LWORD_TO_TIME(in);
TryConvert_LWORD_TO_TIME := TRUE;

END_FUNCTION

// mobject-converters/Converters/LWORD_TO_/TryConvert_LWORD_TO_TOD
FUNCTION TryConvert_LWORD_TO_TOD : BOOL
VAR_INPUT
	in : LWORD;
	out : REFERENCE TO TOD;
END_VAR

IF in > DatatypeLimits.MAX_VALUE_OF_LWORD_WHICH_CAN_BE_HELD_IN_A_TOD THEN
	RETURN;
END_IF

out := LWORD_TO_TOD(in);
TryConvert_LWORD_TO_TOD := TRUE;

END_FUNCTION

// mobject-converters/Converters/LWORD_TO_/TryConvert_LWORD_TO_DT
FUNCTION TryConvert_LWORD_TO_DT : BOOL
VAR_INPUT
	in : LWORD;
	out : REFERENCE TO DT;
END_VAR

IF in > DatatypeLimits.MAX_VALUE_OF_LWORD_WHICH_CAN_BE_HELD_IN_A_DT THEN
	RETURN;
END_IF

out := LWORD_TO_DT(in);
TryConvert_LWORD_TO_DT := TRUE;

END_FUNCTION

// mobject-converters/Converters/LWORD_TO_/TryConvert_LWORD_TO_STRING
FUNCTION TryConvert_LWORD_TO_STRING : BOOL
VAR_INPUT
	in : LWORD;
	out : REFERENCE TO STRING;
END_VAR

out := LWORD_TO_STRING(in);
TryConvert_LWORD_TO_STRING := TRUE;

END_FUNCTION

// mobject-converters/Converters/REAL_TO_/TryConvert_REAL_TO_BOOL
FUNCTION TryConvert_REAL_TO_BOOL : BOOL
VAR_INPUT
	in : REAL;
	out : REFERENCE TO BOOL;
END_VAR

out := REAL_TO_BOOL(in);
TryConvert_REAL_TO_BOOL := TRUE;

END_FUNCTION

// mobject-converters/Converters/REAL_TO_/TryConvert_REAL_TO_BYTE
FUNCTION TryConvert_REAL_TO_BYTE : BOOL
VAR_INPUT
	in : REAL;
	out : REFERENCE TO BYTE;
END_VAR

IF in > DatatypeLimits.MAX_VALUE_OF_REAL_WHICH_CAN_BE_HELD_IN_A_BYTE THEN
	RETURN;
END_IF

IF in < DatatypeLimits.MIN_VALUE_OF_REAL_WHICH_CAN_BE_HELD_IN_A_BYTE THEN
	RETURN;
END_IF

out := REAL_TO_BYTE(in);
TryConvert_REAL_TO_BYTE := TRUE;

END_FUNCTION

// mobject-converters/Converters/REAL_TO_/TryConvert_REAL_TO_DATE
FUNCTION TryConvert_REAL_TO_DATE : BOOL
VAR_INPUT
	in : REAL;
	out : REFERENCE TO DATE;
END_VAR

IF in > DatatypeLimits.MAX_VALUE_OF_REAL_WHICH_CAN_BE_HELD_IN_A_DATE THEN
	RETURN;
END_IF

IF in < DatatypeLimits.MIN_VALUE_OF_REAL_WHICH_CAN_BE_HELD_IN_A_DATE THEN
	RETURN;
END_IF

out := REAL_TO_DATE(in);
TryConvert_REAL_TO_DATE := TRUE;

END_FUNCTION

// mobject-converters/Converters/REAL_TO_/TryConvert_REAL_TO_Destination
FUNCTION TryConvert_REAL_TO_Destination : BOOL
VAR_INPUT
	in : REAL;
	out : ANY;
END_VAR
VAR
	convertResult : BOOL := FALSE;
	convertAddress : PVOID;
	_BOOL : BOOL;
	_BYTE : BYTE;
	_WORD : WORD;
	_DWORD : DWORD;
	_LWORD : LWORD;
	_SINT : SINT;
	_INT : INT;
	_DINT : DINT;
	_LINT : LINT;
	_USINT : USINT;
	_UINT : UINT;
	_UDINT : UDINT;
	_ULINT : ULINT;
	_REAL : REAL;
	_LREAL : LREAL;
	_TIME : TIME;
	_TOD : TOD;
	_DATE : DATE;
	_DT : DT;
	_STRING : STRING;
END_VAR

CASE out.TypeClass OF
	__SYSTEM.TYPE_CLASS.TYPE_BOOL:
	
	convertResult := TryConvert_REAL_TO_BOOL(in, _BOOL);
	IF convertResult THEN
		convertAddress := ADR(_BOOL);
	END_IF
	
	__SYSTEM.TYPE_CLASS.TYPE_BYTE:
	
	convertResult := TryConvert_REAL_TO_BYTE(in, _BYTE);
	IF convertResult THEN
		convertAddress := ADR(_BYTE);
	END_IF
	
	__SYSTEM.TYPE_CLASS.TYPE_WORD:
	
	convertResult := TryConvert_REAL_TO_WORD(in, _WORD);
	IF convertResult THEN
		convertAddress := ADR(_WORD);
	END_IF
	
	__SYSTEM.TYPE_CLASS.TYPE_DWORD:
	
	convertResult := TryConvert_REAL_TO_DWORD(in, _DWORD);
	IF convertResult THEN
		convertAddress := ADR(_DWORD);
	END_IF
	
	__SYSTEM.TYPE_CLASS.TYPE_LWORD:
	
	convertResult := TryConvert_REAL_TO_LWORD(in, _LWORD);
	IF convertResult THEN
		convertAddress := ADR(_LWORD);
	END_IF
	
	__SYSTEM.TYPE_CLASS.TYPE_SINT:
	
	convertResult := TryConvert_REAL_TO_SINT(in, _SINT);
	IF convertResult THEN
		convertAddress := ADR(_SINT);
	END_IF
	
	__SYSTEM.TYPE_CLASS.TYPE_INT:
	
	convertResult := TryConvert_REAL_TO_INT(in, _INT);
	IF convertResult THEN
		convertAddress := ADR(_INT);
	END_IF
	
	__SYSTEM.TYPE_CLASS.TYPE_DINT:
	
	convertResult := TryConvert_REAL_TO_DINT(in, _DINT);
	IF convertResult THEN
		convertAddress := ADR(_DINT);
	END_IF
	
	__SYSTEM.TYPE_CLASS.TYPE_LINT:
	
	convertResult := TryConvert_REAL_TO_LINT(in, _LINT);
	IF convertResult THEN
		convertAddress := ADR(_LINT);
	END_IF
	
	__SYSTEM.TYPE_CLASS.TYPE_USINT:
	
	convertResult := TryConvert_REAL_TO_USINT(in, _USINT);
	IF convertResult THEN
		convertAddress := ADR(_USINT);
	END_IF
	
	__SYSTEM.TYPE_CLASS.TYPE_UINT:
	
	convertResult := TryConvert_REAL_TO_UINT(in, _UINT);
	IF convertResult THEN
		convertAddress := ADR(_UINT);
	END_IF
	
	__SYSTEM.TYPE_CLASS.TYPE_UDINT:
	
	convertResult := TryConvert_REAL_TO_UDINT(in, _UDINT);
	IF convertResult THEN
		convertAddress := ADR(_UDINT);
	END_IF
	
	__SYSTEM.TYPE_CLASS.TYPE_ULINT:
	
	convertResult := TryConvert_REAL_TO_ULINT(in, _ULINT);
	IF convertResult THEN
		convertAddress := ADR(_ULINT);
	END_IF
	
	__SYSTEM.TYPE_CLASS.TYPE_REAL:
	
	convertResult := TryConvert_REAL_TO_REAL(in, _REAL);
	IF convertResult THEN
		convertAddress := ADR(_REAL);
	END_IF
	
	__SYSTEM.TYPE_CLASS.TYPE_LREAL:
	
	convertResult := TryConvert_REAL_TO_LREAL(in, _LREAL);
	IF convertResult THEN
		convertAddress := ADR(_LREAL);
	END_IF
	
	__SYSTEM.TYPE_CLASS.TYPE_TIME:
	
	convertResult := TryConvert_REAL_TO_TIME(in, _TIME);
	IF convertResult THEN
		convertAddress := ADR(_TIME);
	END_IF
	
	__SYSTEM.TYPE_CLASS.TYPE_TIMEOFDAY:
	
	convertResult := TryConvert_REAL_TO_TOD(in, _TOD);
	IF convertResult THEN
		convertAddress := ADR(_TOD);
	END_IF
	
	__SYSTEM.TYPE_CLASS.TYPE_DATE:
	
	convertResult := TryConvert_REAL_TO_DATE(in, _DATE);
	IF convertResult THEN
		convertAddress := ADR(_DATE);
	END_IF
	
	__SYSTEM.TYPE_CLASS.TYPE_DATEANDTIME:
	
	convertResult := TryConvert_REAL_TO_DT(in, _DT);
	IF convertResult THEN
		convertAddress := ADR(_DT);
	END_IF
	
	__SYSTEM.TYPE_CLASS.TYPE_STRING:
	
	convertResult := TryConvert_REAL_TO_STRING(in, _STRING);
	IF convertResult THEN
		convertAddress := ADR(_STRING);
	END_IF
	
END_CASE

IF convertResult THEN
	memcpy(out.pValue,convertAddress,DINT_TO_UDINT(out.diSize));
END_IF

TryConvert_REAL_TO_Destination := convertResult;

END_FUNCTION

// mobject-converters/Converters/REAL_TO_/TryConvert_REAL_TO_WORD
FUNCTION TryConvert_REAL_TO_WORD : BOOL
VAR_INPUT
	in : REAL;
	out : REFERENCE TO WORD;
END_VAR

IF in > DatatypeLimits.MAX_VALUE_OF_REAL_WHICH_CAN_BE_HELD_IN_A_WORD THEN
	RETURN;
END_IF

IF in < DatatypeLimits.MIN_VALUE_OF_REAL_WHICH_CAN_BE_HELD_IN_A_WORD THEN
	RETURN;
END_IF

out := REAL_TO_WORD(in);
TryConvert_REAL_TO_WORD := TRUE;

END_FUNCTION

// mobject-converters/Converters/REAL_TO_/TryConvert_REAL_TO_DWORD
FUNCTION TryConvert_REAL_TO_DWORD : BOOL
VAR_INPUT
	in : REAL;
	out : REFERENCE TO DWORD;
END_VAR

IF in > DatatypeLimits.MAX_VALUE_OF_REAL_WHICH_CAN_BE_HELD_IN_A_DWORD THEN
	RETURN;
END_IF

IF in < DatatypeLimits.MIN_VALUE_OF_REAL_WHICH_CAN_BE_HELD_IN_A_DWORD THEN
	RETURN;
END_IF

out := REAL_TO_DWORD(in);
TryConvert_REAL_TO_DWORD := TRUE;

END_FUNCTION

// mobject-converters/Converters/REAL_TO_/TryConvert_REAL_TO_LWORD
FUNCTION TryConvert_REAL_TO_LWORD : BOOL
VAR_INPUT
	in : REAL;
	out : REFERENCE TO LWORD;
END_VAR

IF in > DatatypeLimits.MAX_VALUE_OF_REAL_WHICH_CAN_BE_HELD_IN_A_LWORD THEN
	RETURN;
END_IF

IF in < DatatypeLimits.MIN_VALUE_OF_REAL_WHICH_CAN_BE_HELD_IN_A_LWORD THEN
	RETURN;
END_IF

out := REAL_TO_LWORD(in);
TryConvert_REAL_TO_LWORD := TRUE;

END_FUNCTION

// mobject-converters/Converters/REAL_TO_/TryConvert_REAL_TO_SINT
FUNCTION TryConvert_REAL_TO_SINT : BOOL
VAR_INPUT
	in : REAL;
	out : REFERENCE TO SINT;
END_VAR

IF in > DatatypeLimits.MAX_VALUE_OF_REAL_WHICH_CAN_BE_HELD_IN_A_SINT THEN
	RETURN;
END_IF

IF in < DatatypeLimits.MIN_VALUE_OF_REAL_WHICH_CAN_BE_HELD_IN_A_SINT THEN
	RETURN;
END_IF

out := REAL_TO_SINT(in);
TryConvert_REAL_TO_SINT := TRUE;

END_FUNCTION

// mobject-converters/Converters/REAL_TO_/TryConvert_REAL_TO_INT
FUNCTION TryConvert_REAL_TO_INT : BOOL
VAR_INPUT
	in : REAL;
	out : REFERENCE TO INT;
END_VAR

IF in > DatatypeLimits.MAX_VALUE_OF_REAL_WHICH_CAN_BE_HELD_IN_A_INT THEN
	RETURN;
END_IF

IF in < DatatypeLimits.MIN_VALUE_OF_REAL_WHICH_CAN_BE_HELD_IN_A_INT THEN
	RETURN;
END_IF

out := REAL_TO_INT(in);
TryConvert_REAL_TO_INT := TRUE;

END_FUNCTION

// mobject-converters/Converters/REAL_TO_/TryConvert_REAL_TO_DINT
FUNCTION TryConvert_REAL_TO_DINT : BOOL
VAR_INPUT
	in : REAL;
	out : REFERENCE TO DINT;
END_VAR

IF in > DatatypeLimits.MAX_VALUE_OF_REAL_WHICH_CAN_BE_HELD_IN_A_DINT THEN
	RETURN;
END_IF

IF in < DatatypeLimits.MIN_VALUE_OF_REAL_WHICH_CAN_BE_HELD_IN_A_DINT THEN
	RETURN;
END_IF

out := REAL_TO_DINT(in);
TryConvert_REAL_TO_DINT := TRUE;

END_FUNCTION

// mobject-converters/Converters/REAL_TO_/TryConvert_REAL_TO_LINT
FUNCTION TryConvert_REAL_TO_LINT : BOOL
VAR_INPUT
	in : REAL;
	out : REFERENCE TO LINT;
END_VAR

IF in > DatatypeLimits.MAX_VALUE_OF_REAL_WHICH_CAN_BE_HELD_IN_A_LINT THEN
	RETURN;
END_IF

IF in < DatatypeLimits.MIN_VALUE_OF_REAL_WHICH_CAN_BE_HELD_IN_A_LINT THEN
	RETURN;
END_IF

out := REAL_TO_LINT(in);
TryConvert_REAL_TO_LINT := TRUE;

END_FUNCTION

// mobject-converters/Converters/REAL_TO_/TryConvert_REAL_TO_USINT
FUNCTION TryConvert_REAL_TO_USINT : BOOL
VAR_INPUT
	in : REAL;
	out : REFERENCE TO USINT;
END_VAR

IF in > DatatypeLimits.MAX_VALUE_OF_REAL_WHICH_CAN_BE_HELD_IN_A_USINT THEN
	RETURN;
END_IF

IF in < DatatypeLimits.MIN_VALUE_OF_REAL_WHICH_CAN_BE_HELD_IN_A_USINT THEN
	RETURN;
END_IF

out := REAL_TO_USINT(in);
TryConvert_REAL_TO_USINT := TRUE;

END_FUNCTION

// mobject-converters/Converters/REAL_TO_/TryConvert_REAL_TO_UINT
FUNCTION TryConvert_REAL_TO_UINT : BOOL
VAR_INPUT
	in : REAL;
	out : REFERENCE TO UINT;
END_VAR

IF in > DatatypeLimits.MAX_VALUE_OF_REAL_WHICH_CAN_BE_HELD_IN_A_UINT THEN
	RETURN;
END_IF

IF in < DatatypeLimits.MIN_VALUE_OF_REAL_WHICH_CAN_BE_HELD_IN_A_UINT THEN
	RETURN;
END_IF

out := REAL_TO_UINT(in);
TryConvert_REAL_TO_UINT := TRUE;

END_FUNCTION

// mobject-converters/Converters/REAL_TO_/TryConvert_REAL_TO_UDINT
FUNCTION TryConvert_REAL_TO_UDINT : BOOL
VAR_INPUT
	in : REAL;
	out : REFERENCE TO UDINT;
END_VAR

IF in > DatatypeLimits.MAX_VALUE_OF_REAL_WHICH_CAN_BE_HELD_IN_A_UDINT THEN
	RETURN;
END_IF

IF in < DatatypeLimits.MIN_VALUE_OF_REAL_WHICH_CAN_BE_HELD_IN_A_UDINT THEN
	RETURN;
END_IF

out := REAL_TO_UDINT(in);
TryConvert_REAL_TO_UDINT := TRUE;

END_FUNCTION

// mobject-converters/Converters/REAL_TO_/TryConvert_REAL_TO_ULINT
FUNCTION TryConvert_REAL_TO_ULINT : BOOL
VAR_INPUT
	in : REAL;
	out : REFERENCE TO ULINT;
END_VAR

IF in > DatatypeLimits.MAX_VALUE_OF_REAL_WHICH_CAN_BE_HELD_IN_A_ULINT THEN
	RETURN;
END_IF

IF in < DatatypeLimits.MIN_VALUE_OF_REAL_WHICH_CAN_BE_HELD_IN_A_ULINT THEN
	RETURN;
END_IF

out := REAL_TO_ULINT(in);
TryConvert_REAL_TO_ULINT := TRUE;

END_FUNCTION

// mobject-converters/Converters/REAL_TO_/TryConvert_REAL_TO_REAL
FUNCTION TryConvert_REAL_TO_REAL : BOOL
VAR_INPUT
	in : REAL;
	out : REFERENCE TO REAL;
END_VAR

out := in;
TryConvert_REAL_TO_REAL := TRUE;

END_FUNCTION

// mobject-converters/Converters/REAL_TO_/TryConvert_REAL_TO_LREAL
FUNCTION TryConvert_REAL_TO_LREAL : BOOL
VAR_INPUT
	in : REAL;
	out : REFERENCE TO LREAL;
END_VAR

out := REAL_TO_LREAL(in);
TryConvert_REAL_TO_LREAL := TRUE;

END_FUNCTION

// mobject-converters/Converters/REAL_TO_/TryConvert_REAL_TO_TIME
FUNCTION TryConvert_REAL_TO_TIME : BOOL
VAR_INPUT
	in : REAL;
	out : REFERENCE TO TIME;
END_VAR

IF in > DatatypeLimits.MAX_VALUE_OF_REAL_WHICH_CAN_BE_HELD_IN_A_TIME THEN
	RETURN;
END_IF

IF in < DatatypeLimits.MIN_VALUE_OF_REAL_WHICH_CAN_BE_HELD_IN_A_TIME THEN
	RETURN;
END_IF

out := REAL_TO_TIME(in);
TryConvert_REAL_TO_TIME := TRUE;

END_FUNCTION

// mobject-converters/Converters/REAL_TO_/TryConvert_REAL_TO_TOD
FUNCTION TryConvert_REAL_TO_TOD : BOOL
VAR_INPUT
	in : REAL;
	out : REFERENCE TO TOD;
END_VAR

IF in > DatatypeLimits.MAX_VALUE_OF_REAL_WHICH_CAN_BE_HELD_IN_A_TOD THEN
	RETURN;
END_IF

IF in < DatatypeLimits.MIN_VALUE_OF_REAL_WHICH_CAN_BE_HELD_IN_A_TOD THEN
	RETURN;
END_IF

out := REAL_TO_TOD(in);
TryConvert_REAL_TO_TOD := TRUE;

END_FUNCTION

// mobject-converters/Converters/REAL_TO_/TryConvert_REAL_TO_DT
FUNCTION TryConvert_REAL_TO_DT : BOOL
VAR_INPUT
	in : REAL;
	out : REFERENCE TO DT;
END_VAR

IF in > DatatypeLimits.MAX_VALUE_OF_REAL_WHICH_CAN_BE_HELD_IN_A_DT THEN
	RETURN;
END_IF

IF in < DatatypeLimits.MIN_VALUE_OF_REAL_WHICH_CAN_BE_HELD_IN_A_DT THEN
	RETURN;
END_IF

out := REAL_TO_DT(in);
TryConvert_REAL_TO_DT := TRUE;

END_FUNCTION

// mobject-converters/Converters/REAL_TO_/TryConvert_REAL_TO_STRING
FUNCTION TryConvert_REAL_TO_STRING : BOOL
VAR_INPUT
	in : REAL;
	out : REFERENCE TO STRING;
END_VAR

out := REAL_TO_STRING(in);
TryConvert_REAL_TO_STRING := TRUE;

END_FUNCTION

// mobject-converters/Converters/SINT_TO_/TryConvert_SINT_TO_BOOL
FUNCTION TryConvert_SINT_TO_BOOL : BOOL
VAR_INPUT
	in : SINT;
	out : REFERENCE TO BOOL;
END_VAR

out := SINT_TO_BOOL(in);
TryConvert_SINT_TO_BOOL := TRUE;

END_FUNCTION

// mobject-converters/Converters/SINT_TO_/TryConvert_SINT_TO_BYTE
FUNCTION TryConvert_SINT_TO_BYTE : BOOL
VAR_INPUT
	in : SINT;
	out : REFERENCE TO BYTE;
END_VAR

IF in < DatatypeLimits.MIN_VALUE_OF_SINT_WHICH_CAN_BE_HELD_IN_A_BYTE THEN
	RETURN;
END_IF

out := SINT_TO_BYTE(in);
TryConvert_SINT_TO_BYTE := TRUE;

END_FUNCTION

// mobject-converters/Converters/SINT_TO_/TryConvert_SINT_TO_DATE
FUNCTION TryConvert_SINT_TO_DATE : BOOL
VAR_INPUT
	in : SINT;
	out : REFERENCE TO DATE;
END_VAR

IF in < DatatypeLimits.MIN_VALUE_OF_SINT_WHICH_CAN_BE_HELD_IN_A_DATE THEN
	RETURN;
END_IF

out := SINT_TO_DATE(in);
TryConvert_SINT_TO_DATE := TRUE;

END_FUNCTION

// mobject-converters/Converters/SINT_TO_/TryConvert_SINT_TO_Destination
FUNCTION TryConvert_SINT_TO_Destination : BOOL
VAR_INPUT
	in : SINT;
	out : ANY;
END_VAR
VAR
	convertResult : BOOL := FALSE;
	convertAddress : PVOID;
	_BOOL : BOOL;
	_BYTE : BYTE;
	_WORD : WORD;
	_DWORD : DWORD;
	_LWORD : LWORD;
	_SINT : SINT;
	_INT : INT;
	_DINT : DINT;
	_LINT : LINT;
	_USINT : USINT;
	_UINT : UINT;
	_UDINT : UDINT;
	_ULINT : ULINT;
	_REAL : REAL;
	_LREAL : LREAL;
	_TIME : TIME;
	_TOD : TOD;
	_DATE : DATE;
	_DT : DT;
	_STRING : STRING;
END_VAR

CASE out.TypeClass OF
	__SYSTEM.TYPE_CLASS.TYPE_BOOL:
	
	convertResult := TryConvert_SINT_TO_BOOL(in, _BOOL);
	IF convertResult THEN
		convertAddress := ADR(_BOOL);
	END_IF
	
	__SYSTEM.TYPE_CLASS.TYPE_BYTE:
	
	convertResult := TryConvert_SINT_TO_BYTE(in, _BYTE);
	IF convertResult THEN
		convertAddress := ADR(_BYTE);
	END_IF
	
	__SYSTEM.TYPE_CLASS.TYPE_WORD:
	
	convertResult := TryConvert_SINT_TO_WORD(in, _WORD);
	IF convertResult THEN
		convertAddress := ADR(_WORD);
	END_IF
	
	__SYSTEM.TYPE_CLASS.TYPE_DWORD:
	
	convertResult := TryConvert_SINT_TO_DWORD(in, _DWORD);
	IF convertResult THEN
		convertAddress := ADR(_DWORD);
	END_IF
	
	__SYSTEM.TYPE_CLASS.TYPE_LWORD:
	
	convertResult := TryConvert_SINT_TO_LWORD(in, _LWORD);
	IF convertResult THEN
		convertAddress := ADR(_LWORD);
	END_IF
	
	__SYSTEM.TYPE_CLASS.TYPE_SINT:
	
	convertResult := TryConvert_SINT_TO_SINT(in, _SINT);
	IF convertResult THEN
		convertAddress := ADR(_SINT);
	END_IF
	
	__SYSTEM.TYPE_CLASS.TYPE_INT:
	
	convertResult := TryConvert_SINT_TO_INT(in, _INT);
	IF convertResult THEN
		convertAddress := ADR(_INT);
	END_IF
	
	__SYSTEM.TYPE_CLASS.TYPE_DINT:
	
	convertResult := TryConvert_SINT_TO_DINT(in, _DINT);
	IF convertResult THEN
		convertAddress := ADR(_DINT);
	END_IF
	
	__SYSTEM.TYPE_CLASS.TYPE_LINT:
	
	convertResult := TryConvert_SINT_TO_LINT(in, _LINT);
	IF convertResult THEN
		convertAddress := ADR(_LINT);
	END_IF
	
	__SYSTEM.TYPE_CLASS.TYPE_USINT:
	
	convertResult := TryConvert_SINT_TO_USINT(in, _USINT);
	IF convertResult THEN
		convertAddress := ADR(_USINT);
	END_IF
	
	__SYSTEM.TYPE_CLASS.TYPE_UINT:
	
	convertResult := TryConvert_SINT_TO_UINT(in, _UINT);
	IF convertResult THEN
		convertAddress := ADR(_UINT);
	END_IF
	
	__SYSTEM.TYPE_CLASS.TYPE_UDINT:
	
	convertResult := TryConvert_SINT_TO_UDINT(in, _UDINT);
	IF convertResult THEN
		convertAddress := ADR(_UDINT);
	END_IF
	
	__SYSTEM.TYPE_CLASS.TYPE_ULINT:
	
	convertResult := TryConvert_SINT_TO_ULINT(in, _ULINT);
	IF convertResult THEN
		convertAddress := ADR(_ULINT);
	END_IF
	
	__SYSTEM.TYPE_CLASS.TYPE_REAL:
	
	convertResult := TryConvert_SINT_TO_REAL(in, _REAL);
	IF convertResult THEN
		convertAddress := ADR(_REAL);
	END_IF
	
	__SYSTEM.TYPE_CLASS.TYPE_LREAL:
	
	convertResult := TryConvert_SINT_TO_LREAL(in, _LREAL);
	IF convertResult THEN
		convertAddress := ADR(_LREAL);
	END_IF
	
	__SYSTEM.TYPE_CLASS.TYPE_TIME:
	
	convertResult := TryConvert_SINT_TO_TIME(in, _TIME);
	IF convertResult THEN
		convertAddress := ADR(_TIME);
	END_IF
	
	__SYSTEM.TYPE_CLASS.TYPE_TIMEOFDAY:
	
	convertResult := TryConvert_SINT_TO_TOD(in, _TOD);
	IF convertResult THEN
		convertAddress := ADR(_TOD);
	END_IF
	
	__SYSTEM.TYPE_CLASS.TYPE_DATE:
	
	convertResult := TryConvert_SINT_TO_DATE(in, _DATE);
	IF convertResult THEN
		convertAddress := ADR(_DATE);
	END_IF
	
	__SYSTEM.TYPE_CLASS.TYPE_DATEANDTIME:
	
	convertResult := TryConvert_SINT_TO_DT(in, _DT);
	IF convertResult THEN
		convertAddress := ADR(_DT);
	END_IF
	
	__SYSTEM.TYPE_CLASS.TYPE_STRING:
	
	convertResult := TryConvert_SINT_TO_STRING(in, _STRING);
	IF convertResult THEN
		convertAddress := ADR(_STRING);
	END_IF
	
END_CASE

IF convertResult THEN
	memcpy(out.pValue,convertAddress,DINT_TO_UDINT(out.diSize));
END_IF

TryConvert_SINT_TO_Destination := convertResult;

END_FUNCTION

// mobject-converters/Converters/SINT_TO_/TryConvert_SINT_TO_WORD
FUNCTION TryConvert_SINT_TO_WORD : BOOL
VAR_INPUT
	in : SINT;
	out : REFERENCE TO WORD;
END_VAR

IF in < DatatypeLimits.MIN_VALUE_OF_SINT_WHICH_CAN_BE_HELD_IN_A_WORD THEN
	RETURN;
END_IF

out := SINT_TO_WORD(in);
TryConvert_SINT_TO_WORD := TRUE;

END_FUNCTION

// mobject-converters/Converters/SINT_TO_/TryConvert_SINT_TO_DWORD
FUNCTION TryConvert_SINT_TO_DWORD : BOOL
VAR_INPUT
	in : SINT;
	out : REFERENCE TO DWORD;
END_VAR

IF in < DatatypeLimits.MIN_VALUE_OF_SINT_WHICH_CAN_BE_HELD_IN_A_DWORD THEN
	RETURN;
END_IF

out := SINT_TO_DWORD(in);
TryConvert_SINT_TO_DWORD := TRUE;

END_FUNCTION

// mobject-converters/Converters/SINT_TO_/TryConvert_SINT_TO_LWORD
FUNCTION TryConvert_SINT_TO_LWORD : BOOL
VAR_INPUT
	in : SINT;
	out : REFERENCE TO LWORD;
END_VAR

IF in < DatatypeLimits.MIN_VALUE_OF_SINT_WHICH_CAN_BE_HELD_IN_A_LWORD THEN
	RETURN;
END_IF

out := SINT_TO_LWORD(in);
TryConvert_SINT_TO_LWORD := TRUE;

END_FUNCTION

// mobject-converters/Converters/SINT_TO_/TryConvert_SINT_TO_SINT
FUNCTION TryConvert_SINT_TO_SINT : BOOL
VAR_INPUT
	in : SINT;
	out : REFERENCE TO SINT;
END_VAR

out := in;
TryConvert_SINT_TO_SINT := TRUE;

END_FUNCTION

// mobject-converters/Converters/SINT_TO_/TryConvert_SINT_TO_INT
FUNCTION TryConvert_SINT_TO_INT : BOOL
VAR_INPUT
	in : SINT;
	out : REFERENCE TO INT;
END_VAR

out := SINT_TO_INT(in);
TryConvert_SINT_TO_INT := TRUE;

END_FUNCTION

// mobject-converters/Converters/SINT_TO_/TryConvert_SINT_TO_DINT
FUNCTION TryConvert_SINT_TO_DINT : BOOL
VAR_INPUT
	in : SINT;
	out : REFERENCE TO DINT;
END_VAR

out := SINT_TO_DINT(in);
TryConvert_SINT_TO_DINT := TRUE;

END_FUNCTION

// mobject-converters/Converters/SINT_TO_/TryConvert_SINT_TO_LINT
FUNCTION TryConvert_SINT_TO_LINT : BOOL
VAR_INPUT
	in : SINT;
	out : REFERENCE TO LINT;
END_VAR

out := SINT_TO_LINT(in);
TryConvert_SINT_TO_LINT := TRUE;

END_FUNCTION

// mobject-converters/Converters/SINT_TO_/TryConvert_SINT_TO_USINT
FUNCTION TryConvert_SINT_TO_USINT : BOOL
VAR_INPUT
	in : SINT;
	out : REFERENCE TO USINT;
END_VAR

IF in < DatatypeLimits.MIN_VALUE_OF_SINT_WHICH_CAN_BE_HELD_IN_A_USINT THEN
	RETURN;
END_IF

out := SINT_TO_USINT(in);
TryConvert_SINT_TO_USINT := TRUE;

END_FUNCTION

// mobject-converters/Converters/SINT_TO_/TryConvert_SINT_TO_UINT
FUNCTION TryConvert_SINT_TO_UINT : BOOL
VAR_INPUT
	in : SINT;
	out : REFERENCE TO UINT;
END_VAR

IF in < DatatypeLimits.MIN_VALUE_OF_SINT_WHICH_CAN_BE_HELD_IN_A_UINT THEN
	RETURN;
END_IF

out := SINT_TO_UINT(in);
TryConvert_SINT_TO_UINT := TRUE;

END_FUNCTION

// mobject-converters/Converters/SINT_TO_/TryConvert_SINT_TO_UDINT
FUNCTION TryConvert_SINT_TO_UDINT : BOOL
VAR_INPUT
	in : SINT;
	out : REFERENCE TO UDINT;
END_VAR

IF in < DatatypeLimits.MIN_VALUE_OF_SINT_WHICH_CAN_BE_HELD_IN_A_UDINT THEN
	RETURN;
END_IF

out := SINT_TO_UDINT(in);
TryConvert_SINT_TO_UDINT := TRUE;

END_FUNCTION

// mobject-converters/Converters/SINT_TO_/TryConvert_SINT_TO_ULINT
FUNCTION TryConvert_SINT_TO_ULINT : BOOL
VAR_INPUT
	in : SINT;
	out : REFERENCE TO ULINT;
END_VAR

IF in < DatatypeLimits.MIN_VALUE_OF_SINT_WHICH_CAN_BE_HELD_IN_A_ULINT THEN
	RETURN;
END_IF

out := SINT_TO_ULINT(in);
TryConvert_SINT_TO_ULINT := TRUE;

END_FUNCTION

// mobject-converters/Converters/SINT_TO_/TryConvert_SINT_TO_REAL
FUNCTION TryConvert_SINT_TO_REAL : BOOL
VAR_INPUT
	in : SINT;
	out : REFERENCE TO REAL;
END_VAR

out := SINT_TO_REAL(in);
TryConvert_SINT_TO_REAL := TRUE;

END_FUNCTION

// mobject-converters/Converters/SINT_TO_/TryConvert_SINT_TO_LREAL
FUNCTION TryConvert_SINT_TO_LREAL : BOOL
VAR_INPUT
	in : SINT;
	out : REFERENCE TO LREAL;
END_VAR

out := SINT_TO_LREAL(in);
TryConvert_SINT_TO_LREAL := TRUE;

END_FUNCTION

// mobject-converters/Converters/SINT_TO_/TryConvert_SINT_TO_TIME
FUNCTION TryConvert_SINT_TO_TIME : BOOL
VAR_INPUT
	in : SINT;
	out : REFERENCE TO TIME;
END_VAR

IF in < DatatypeLimits.MIN_VALUE_OF_SINT_WHICH_CAN_BE_HELD_IN_A_TIME THEN
	RETURN;
END_IF

out := SINT_TO_TIME(in);
TryConvert_SINT_TO_TIME := TRUE;

END_FUNCTION

// mobject-converters/Converters/SINT_TO_/TryConvert_SINT_TO_TOD
FUNCTION TryConvert_SINT_TO_TOD : BOOL
VAR_INPUT
	in : SINT;
	out : REFERENCE TO TOD;
END_VAR

IF in < DatatypeLimits.MIN_VALUE_OF_SINT_WHICH_CAN_BE_HELD_IN_A_TOD THEN
	RETURN;
END_IF

out := SINT_TO_TOD(in);
TryConvert_SINT_TO_TOD := TRUE;

END_FUNCTION

// mobject-converters/Converters/SINT_TO_/TryConvert_SINT_TO_DT
FUNCTION TryConvert_SINT_TO_DT : BOOL
VAR_INPUT
	in : SINT;
	out : REFERENCE TO DT;
END_VAR

IF in < DatatypeLimits.MIN_VALUE_OF_SINT_WHICH_CAN_BE_HELD_IN_A_DT THEN
	RETURN;
END_IF

out := SINT_TO_DT(in);
TryConvert_SINT_TO_DT := TRUE;

END_FUNCTION

// mobject-converters/Converters/SINT_TO_/TryConvert_SINT_TO_STRING
FUNCTION TryConvert_SINT_TO_STRING : BOOL
VAR_INPUT
	in : SINT;
	out : REFERENCE TO STRING;
END_VAR

out := SINT_TO_STRING(in);
TryConvert_SINT_TO_STRING := TRUE;

END_FUNCTION

// mobject-converters/Converters/STRING_TO_/TryConvert_STRING_TO_BOOL
FUNCTION TryConvert_STRING_TO_BOOL : BOOL
VAR_INPUT
	in : STRING;
	out : REFERENCE TO BOOL;
END_VAR

out := STRING_TO_BOOL(in);
TryConvert_STRING_TO_BOOL := TRUE;

END_FUNCTION

// mobject-converters/Converters/STRING_TO_/TryConvert_STRING_TO_BYTE
FUNCTION TryConvert_STRING_TO_BYTE : BOOL
VAR_INPUT
	in : STRING;
	out : REFERENCE TO BYTE;
END_VAR

IF in <> BYTE_TO_STRING(STRING_TO_BYTE(in)) THEN
	RETURN;
END_IF

out := STRING_TO_BYTE(in);
TryConvert_STRING_TO_BYTE := TRUE;

END_FUNCTION

// mobject-converters/Converters/STRING_TO_/TryConvert_STRING_TO_DATE
FUNCTION TryConvert_STRING_TO_DATE : BOOL
VAR_INPUT
	in : STRING;
	out : REFERENCE TO DATE;
END_VAR

IF in <> DATE_TO_STRING(STRING_TO_DATE(in)) THEN
	RETURN;
END_IF

out := STRING_TO_DATE(in);
TryConvert_STRING_TO_DATE := TRUE;

END_FUNCTION

// mobject-converters/Converters/STRING_TO_/TryConvert_STRING_TO_Destination
FUNCTION TryConvert_STRING_TO_Destination : BOOL
VAR_INPUT
	in : STRING;
	out : ANY;
END_VAR
VAR
	convertResult : BOOL := FALSE;
	convertAddress : PVOID;
	_BOOL : BOOL;
	_BYTE : BYTE;
	_WORD : WORD;
	_DWORD : DWORD;
	_LWORD : LWORD;
	_SINT : SINT;
	_INT : INT;
	_DINT : DINT;
	_LINT : LINT;
	_USINT : USINT;
	_UINT : UINT;
	_UDINT : UDINT;
	_ULINT : ULINT;
	_REAL : REAL;
	_LREAL : LREAL;
	_TIME : TIME;
	_TOD : TOD;
	_DATE : DATE;
	_DT : DT;
	_STRING : STRING;
END_VAR

CASE out.TypeClass OF
	__SYSTEM.TYPE_CLASS.TYPE_BOOL:
	
	convertResult := TryConvert_STRING_TO_BOOL(in, _BOOL);
	IF convertResult THEN
		convertAddress := ADR(_BOOL);
	END_IF
	
	__SYSTEM.TYPE_CLASS.TYPE_BYTE:
	
	convertResult := TryConvert_STRING_TO_BYTE(in, _BYTE);
	IF convertResult THEN
		convertAddress := ADR(_BYTE);
	END_IF
	
	__SYSTEM.TYPE_CLASS.TYPE_WORD:
	
	convertResult := TryConvert_STRING_TO_WORD(in, _WORD);
	IF convertResult THEN
		convertAddress := ADR(_WORD);
	END_IF
	
	__SYSTEM.TYPE_CLASS.TYPE_DWORD:
	
	convertResult := TryConvert_STRING_TO_DWORD(in, _DWORD);
	IF convertResult THEN
		convertAddress := ADR(_DWORD);
	END_IF
	
	__SYSTEM.TYPE_CLASS.TYPE_LWORD:
	
	convertResult := TryConvert_STRING_TO_LWORD(in, _LWORD);
	IF convertResult THEN
		convertAddress := ADR(_LWORD);
	END_IF
	
	__SYSTEM.TYPE_CLASS.TYPE_SINT:
	
	convertResult := TryConvert_STRING_TO_SINT(in, _SINT);
	IF convertResult THEN
		convertAddress := ADR(_SINT);
	END_IF
	
	__SYSTEM.TYPE_CLASS.TYPE_INT:
	
	convertResult := TryConvert_STRING_TO_INT(in, _INT);
	IF convertResult THEN
		convertAddress := ADR(_INT);
	END_IF
	
	__SYSTEM.TYPE_CLASS.TYPE_DINT:
	
	convertResult := TryConvert_STRING_TO_DINT(in, _DINT);
	IF convertResult THEN
		convertAddress := ADR(_DINT);
	END_IF
	
	__SYSTEM.TYPE_CLASS.TYPE_LINT:
	
	convertResult := TryConvert_STRING_TO_LINT(in, _LINT);
	IF convertResult THEN
		convertAddress := ADR(_LINT);
	END_IF
	
	__SYSTEM.TYPE_CLASS.TYPE_USINT:
	
	convertResult := TryConvert_STRING_TO_USINT(in, _USINT);
	IF convertResult THEN
		convertAddress := ADR(_USINT);
	END_IF
	
	__SYSTEM.TYPE_CLASS.TYPE_UINT:
	
	convertResult := TryConvert_STRING_TO_UINT(in, _UINT);
	IF convertResult THEN
		convertAddress := ADR(_UINT);
	END_IF
	
	__SYSTEM.TYPE_CLASS.TYPE_UDINT:
	
	convertResult := TryConvert_STRING_TO_UDINT(in, _UDINT);
	IF convertResult THEN
		convertAddress := ADR(_UDINT);
	END_IF
	
	__SYSTEM.TYPE_CLASS.TYPE_ULINT:
	
	convertResult := TryConvert_STRING_TO_ULINT(in, _ULINT);
	IF convertResult THEN
		convertAddress := ADR(_ULINT);
	END_IF
	
	__SYSTEM.TYPE_CLASS.TYPE_REAL:
	
	convertResult := TryConvert_STRING_TO_REAL(in, _REAL);
	IF convertResult THEN
		convertAddress := ADR(_REAL);
	END_IF
	
	__SYSTEM.TYPE_CLASS.TYPE_LREAL:
	
	convertResult := TryConvert_STRING_TO_LREAL(in, _LREAL);
	IF convertResult THEN
		convertAddress := ADR(_LREAL);
	END_IF
	
	__SYSTEM.TYPE_CLASS.TYPE_TIME:
	
	convertResult := TryConvert_STRING_TO_TIME(in, _TIME);
	IF convertResult THEN
		convertAddress := ADR(_TIME);
	END_IF
	
	__SYSTEM.TYPE_CLASS.TYPE_TIMEOFDAY:
	
	convertResult := TryConvert_STRING_TO_TOD(in, _TOD);
	IF convertResult THEN
		convertAddress := ADR(_TOD);
	END_IF
	
	__SYSTEM.TYPE_CLASS.TYPE_DATE:
	
	convertResult := TryConvert_STRING_TO_DATE(in, _DATE);
	IF convertResult THEN
		convertAddress := ADR(_DATE);
	END_IF
	
	__SYSTEM.TYPE_CLASS.TYPE_DATEANDTIME:
	
	convertResult := TryConvert_STRING_TO_DT(in, _DT);
	IF convertResult THEN
		convertAddress := ADR(_DT);
	END_IF
	
	__SYSTEM.TYPE_CLASS.TYPE_STRING:
	
	convertResult := TryConvert_STRING_TO_STRING(in, _STRING);
	IF convertResult THEN
		convertAddress := ADR(_STRING);
	END_IF
	
END_CASE

IF convertResult THEN
	memcpy(out.pValue,convertAddress,DINT_TO_UDINT(out.diSize));
END_IF

TryConvert_STRING_TO_Destination := convertResult;

END_FUNCTION

// mobject-converters/Converters/STRING_TO_/TryConvert_STRING_TO_WORD
FUNCTION TryConvert_STRING_TO_WORD : BOOL
VAR_INPUT
	in : STRING;
	out : REFERENCE TO WORD;
END_VAR

IF in <> WORD_TO_STRING(STRING_TO_WORD(in)) THEN
	RETURN;
END_IF

out := STRING_TO_WORD(in);
TryConvert_STRING_TO_WORD := TRUE;

END_FUNCTION

// mobject-converters/Converters/STRING_TO_/TryConvert_STRING_TO_DWORD
FUNCTION TryConvert_STRING_TO_DWORD : BOOL
VAR_INPUT
	in : STRING;
	out : REFERENCE TO DWORD;
END_VAR

IF in <> DWORD_TO_STRING(STRING_TO_DWORD(in)) THEN
	RETURN;
END_IF

out := STRING_TO_DWORD(in);
TryConvert_STRING_TO_DWORD := TRUE;

END_FUNCTION

// mobject-converters/Converters/STRING_TO_/TryConvert_STRING_TO_LWORD
FUNCTION TryConvert_STRING_TO_LWORD : BOOL
VAR_INPUT
	in : STRING;
	out : REFERENCE TO LWORD;
END_VAR

IF in <> LWORD_TO_STRING(STRING_TO_LWORD(in)) THEN
	RETURN;
END_IF

out := STRING_TO_LWORD(in);
TryConvert_STRING_TO_LWORD := TRUE;

END_FUNCTION

// mobject-converters/Converters/STRING_TO_/TryConvert_STRING_TO_SINT
FUNCTION TryConvert_STRING_TO_SINT : BOOL
VAR_INPUT
	in : STRING;
	out : REFERENCE TO SINT;
END_VAR

IF in <> SINT_TO_STRING(STRING_TO_SINT(in)) THEN
	RETURN;
END_IF

out := STRING_TO_SINT(in);
TryConvert_STRING_TO_SINT := TRUE;

END_FUNCTION

// mobject-converters/Converters/STRING_TO_/TryConvert_STRING_TO_INT
FUNCTION TryConvert_STRING_TO_INT : BOOL
VAR_INPUT
	in : STRING;
	out : REFERENCE TO INT;
END_VAR

IF in <> INT_TO_STRING(STRING_TO_INT(in)) THEN
	RETURN;
END_IF

out := STRING_TO_INT(in);
TryConvert_STRING_TO_INT := TRUE;

END_FUNCTION

// mobject-converters/Converters/STRING_TO_/TryConvert_STRING_TO_DINT
FUNCTION TryConvert_STRING_TO_DINT : BOOL
VAR_INPUT
	in : STRING;
	out : REFERENCE TO DINT;
END_VAR

IF in <> DINT_TO_STRING(STRING_TO_DINT(in)) THEN
	RETURN;
END_IF

out := STRING_TO_DINT(in);
TryConvert_STRING_TO_DINT := TRUE;

END_FUNCTION

// mobject-converters/Converters/STRING_TO_/TryConvert_STRING_TO_LINT
FUNCTION TryConvert_STRING_TO_LINT : BOOL
VAR_INPUT
	in : STRING;
	out : REFERENCE TO LINT;
END_VAR

IF in <> LINT_TO_STRING(STRING_TO_LINT(in)) THEN
	RETURN;
END_IF

out := STRING_TO_LINT(in);
TryConvert_STRING_TO_LINT := TRUE;

END_FUNCTION

// mobject-converters/Converters/STRING_TO_/TryConvert_STRING_TO_USINT
FUNCTION TryConvert_STRING_TO_USINT : BOOL
VAR_INPUT
	in : STRING;
	out : REFERENCE TO USINT;
END_VAR

IF in <> USINT_TO_STRING(STRING_TO_USINT(in)) THEN
	RETURN;
END_IF

out := STRING_TO_USINT(in);
TryConvert_STRING_TO_USINT := TRUE;

END_FUNCTION

// mobject-converters/Converters/STRING_TO_/TryConvert_STRING_TO_UINT
FUNCTION TryConvert_STRING_TO_UINT : BOOL
VAR_INPUT
	in : STRING;
	out : REFERENCE TO UINT;
END_VAR

IF in <> UINT_TO_STRING(STRING_TO_UINT(in)) THEN
	RETURN;
END_IF

out := STRING_TO_UINT(in);
TryConvert_STRING_TO_UINT := TRUE;

END_FUNCTION

// mobject-converters/Converters/STRING_TO_/TryConvert_STRING_TO_UDINT
FUNCTION TryConvert_STRING_TO_UDINT : BOOL
VAR_INPUT
	in : STRING;
	out : REFERENCE TO UDINT;
END_VAR

IF in <> UDINT_TO_STRING(STRING_TO_UDINT(in)) THEN
	RETURN;
END_IF

out := STRING_TO_UDINT(in);
TryConvert_STRING_TO_UDINT := TRUE;

END_FUNCTION

// mobject-converters/Converters/STRING_TO_/TryConvert_STRING_TO_ULINT
FUNCTION TryConvert_STRING_TO_ULINT : BOOL
VAR_INPUT
	in : STRING;
	out : REFERENCE TO ULINT;
END_VAR

IF in <> ULINT_TO_STRING(STRING_TO_ULINT(in)) THEN
	RETURN;
END_IF

out := STRING_TO_ULINT(in);
TryConvert_STRING_TO_ULINT := TRUE;

END_FUNCTION

// mobject-converters/Converters/STRING_TO_/TryConvert_STRING_TO_REAL
FUNCTION TryConvert_STRING_TO_REAL : BOOL
VAR_INPUT
	in : STRING;
	out : REFERENCE TO REAL;
END_VAR

IF in <> REAL_TO_STRING(STRING_TO_REAL(in)) THEN
	RETURN;
END_IF

out := STRING_TO_REAL(in);
TryConvert_STRING_TO_REAL := TRUE;

END_FUNCTION

// mobject-converters/Converters/STRING_TO_/TryConvert_STRING_TO_LREAL
FUNCTION TryConvert_STRING_TO_LREAL : BOOL
VAR_INPUT
	in : STRING;
	out : REFERENCE TO LREAL;
END_VAR

IF in <> LREAL_TO_STRING(STRING_TO_LREAL(in)) THEN
	RETURN;
END_IF

out := STRING_TO_LREAL(in);
TryConvert_STRING_TO_LREAL := TRUE;

END_FUNCTION

// mobject-converters/Converters/STRING_TO_/TryConvert_STRING_TO_TIME
FUNCTION TryConvert_STRING_TO_TIME : BOOL
VAR_INPUT
	in : STRING;
	out : REFERENCE TO TIME;
END_VAR

IF in <> TIME_TO_STRING(STRING_TO_TIME(in)) THEN
	RETURN;
END_IF

out := STRING_TO_TIME(in);
TryConvert_STRING_TO_TIME := TRUE;

END_FUNCTION

// mobject-converters/Converters/STRING_TO_/TryConvert_STRING_TO_TOD
FUNCTION TryConvert_STRING_TO_TOD : BOOL
VAR_INPUT
	in : STRING;
	out : REFERENCE TO TOD;
END_VAR

IF in <> TOD_TO_STRING(STRING_TO_TOD(in)) THEN
	RETURN;
END_IF

out := STRING_TO_TOD(in);
TryConvert_STRING_TO_TOD := TRUE;

END_FUNCTION

// mobject-converters/Converters/STRING_TO_/TryConvert_STRING_TO_DT
FUNCTION TryConvert_STRING_TO_DT : BOOL
VAR_INPUT
	in : STRING;
	out : REFERENCE TO DT;
END_VAR

IF in <> DT_TO_STRING(STRING_TO_DT(in)) THEN
	RETURN;
END_IF

out := STRING_TO_DT(in);
TryConvert_STRING_TO_DT := TRUE;

END_FUNCTION

// mobject-converters/Converters/STRING_TO_/TryConvert_STRING_TO_STRING
FUNCTION TryConvert_STRING_TO_STRING : BOOL
VAR_INPUT
	in : STRING;
	out : REFERENCE TO STRING;
END_VAR

out := in;
TryConvert_STRING_TO_STRING := TRUE;

END_FUNCTION

// mobject-converters/Converters/TIME_TO_/TryConvert_TIME_TO_BOOL
FUNCTION TryConvert_TIME_TO_BOOL : BOOL
VAR_INPUT
	in : TIME;
	out : REFERENCE TO BOOL;
END_VAR

out := TIME_TO_BOOL(in);
TryConvert_TIME_TO_BOOL := TRUE;

END_FUNCTION

// mobject-converters/Converters/TIME_TO_/TryConvert_TIME_TO_BYTE
FUNCTION TryConvert_TIME_TO_BYTE : BOOL
VAR_INPUT
	in : TIME;
	out : REFERENCE TO BYTE;
END_VAR

IF in > DatatypeLimits.MAX_VALUE_OF_TIME_WHICH_CAN_BE_HELD_IN_A_BYTE THEN
	RETURN;
END_IF

out := TIME_TO_BYTE(in);
TryConvert_TIME_TO_BYTE := TRUE;

END_FUNCTION

// mobject-converters/Converters/TIME_TO_/TryConvert_TIME_TO_DATE
FUNCTION TryConvert_TIME_TO_DATE : BOOL
VAR_INPUT
	in : TIME;
	out : REFERENCE TO DATE;
END_VAR

out := TIME_TO_DATE(in);
TryConvert_TIME_TO_DATE := TRUE;

END_FUNCTION

// mobject-converters/Converters/TIME_TO_/TryConvert_TIME_TO_Destination
FUNCTION TryConvert_TIME_TO_Destination : BOOL
VAR_INPUT
	in : TIME;
	out : ANY;
END_VAR
VAR
	convertResult : BOOL := FALSE;
	convertAddress : PVOID;
	_BOOL : BOOL;
	_BYTE : BYTE;
	_WORD : WORD;
	_DWORD : DWORD;
	_LWORD : LWORD;
	_SINT : SINT;
	_INT : INT;
	_DINT : DINT;
	_LINT : LINT;
	_USINT : USINT;
	_UINT : UINT;
	_UDINT : UDINT;
	_ULINT : ULINT;
	_REAL : REAL;
	_LREAL : LREAL;
	_TIME : TIME;
	_TOD : TOD;
	_DATE : DATE;
	_DT : DT;
	_STRING : STRING;
END_VAR

CASE out.TypeClass OF
	__SYSTEM.TYPE_CLASS.TYPE_BOOL:
	
	convertResult := TryConvert_TIME_TO_BOOL(in, _BOOL);
	IF convertResult THEN
		convertAddress := ADR(_BOOL);
	END_IF
	
	__SYSTEM.TYPE_CLASS.TYPE_BYTE:
	
	convertResult := TryConvert_TIME_TO_BYTE(in, _BYTE);
	IF convertResult THEN
		convertAddress := ADR(_BYTE);
	END_IF
	
	__SYSTEM.TYPE_CLASS.TYPE_WORD:
	
	convertResult := TryConvert_TIME_TO_WORD(in, _WORD);
	IF convertResult THEN
		convertAddress := ADR(_WORD);
	END_IF
	
	__SYSTEM.TYPE_CLASS.TYPE_DWORD:
	
	convertResult := TryConvert_TIME_TO_DWORD(in, _DWORD);
	IF convertResult THEN
		convertAddress := ADR(_DWORD);
	END_IF
	
	__SYSTEM.TYPE_CLASS.TYPE_LWORD:
	
	convertResult := TryConvert_TIME_TO_LWORD(in, _LWORD);
	IF convertResult THEN
		convertAddress := ADR(_LWORD);
	END_IF
	
	__SYSTEM.TYPE_CLASS.TYPE_SINT:
	
	convertResult := TryConvert_TIME_TO_SINT(in, _SINT);
	IF convertResult THEN
		convertAddress := ADR(_SINT);
	END_IF
	
	__SYSTEM.TYPE_CLASS.TYPE_INT:
	
	convertResult := TryConvert_TIME_TO_INT(in, _INT);
	IF convertResult THEN
		convertAddress := ADR(_INT);
	END_IF
	
	__SYSTEM.TYPE_CLASS.TYPE_DINT:
	
	convertResult := TryConvert_TIME_TO_DINT(in, _DINT);
	IF convertResult THEN
		convertAddress := ADR(_DINT);
	END_IF
	
	__SYSTEM.TYPE_CLASS.TYPE_LINT:
	
	convertResult := TryConvert_TIME_TO_LINT(in, _LINT);
	IF convertResult THEN
		convertAddress := ADR(_LINT);
	END_IF
	
	__SYSTEM.TYPE_CLASS.TYPE_USINT:
	
	convertResult := TryConvert_TIME_TO_USINT(in, _USINT);
	IF convertResult THEN
		convertAddress := ADR(_USINT);
	END_IF
	
	__SYSTEM.TYPE_CLASS.TYPE_UINT:
	
	convertResult := TryConvert_TIME_TO_UINT(in, _UINT);
	IF convertResult THEN
		convertAddress := ADR(_UINT);
	END_IF
	
	__SYSTEM.TYPE_CLASS.TYPE_UDINT:
	
	convertResult := TryConvert_TIME_TO_UDINT(in, _UDINT);
	IF convertResult THEN
		convertAddress := ADR(_UDINT);
	END_IF
	
	__SYSTEM.TYPE_CLASS.TYPE_ULINT:
	
	convertResult := TryConvert_TIME_TO_ULINT(in, _ULINT);
	IF convertResult THEN
		convertAddress := ADR(_ULINT);
	END_IF
	
	__SYSTEM.TYPE_CLASS.TYPE_REAL:
	
	convertResult := TryConvert_TIME_TO_REAL(in, _REAL);
	IF convertResult THEN
		convertAddress := ADR(_REAL);
	END_IF
	
	__SYSTEM.TYPE_CLASS.TYPE_LREAL:
	
	convertResult := TryConvert_TIME_TO_LREAL(in, _LREAL);
	IF convertResult THEN
		convertAddress := ADR(_LREAL);
	END_IF
	
	__SYSTEM.TYPE_CLASS.TYPE_TIME:
	
	convertResult := TryConvert_TIME_TO_TIME(in, _TIME);
	IF convertResult THEN
		convertAddress := ADR(_TIME);
	END_IF
	
	__SYSTEM.TYPE_CLASS.TYPE_TIMEOFDAY:
	
	convertResult := TryConvert_TIME_TO_TOD(in, _TOD);
	IF convertResult THEN
		convertAddress := ADR(_TOD);
	END_IF
	
	__SYSTEM.TYPE_CLASS.TYPE_DATE:
	
	convertResult := TryConvert_TIME_TO_DATE(in, _DATE);
	IF convertResult THEN
		convertAddress := ADR(_DATE);
	END_IF
	
	__SYSTEM.TYPE_CLASS.TYPE_DATEANDTIME:
	
	convertResult := TryConvert_TIME_TO_DT(in, _DT);
	IF convertResult THEN
		convertAddress := ADR(_DT);
	END_IF
	
	__SYSTEM.TYPE_CLASS.TYPE_STRING:
	
	convertResult := TryConvert_TIME_TO_STRING(in, _STRING);
	IF convertResult THEN
		convertAddress := ADR(_STRING);
	END_IF
	
END_CASE

IF convertResult THEN
	memcpy(out.pValue,convertAddress,DINT_TO_UDINT(out.diSize));
END_IF

TryConvert_TIME_TO_Destination := convertResult;

END_FUNCTION

// mobject-converters/Converters/TIME_TO_/TryConvert_TIME_TO_WORD
FUNCTION TryConvert_TIME_TO_WORD : BOOL
VAR_INPUT
	in : TIME;
	out : REFERENCE TO WORD;
END_VAR

IF in > DatatypeLimits.MAX_VALUE_OF_TIME_WHICH_CAN_BE_HELD_IN_A_WORD THEN
	RETURN;
END_IF

out := TIME_TO_WORD(in);
TryConvert_TIME_TO_WORD := TRUE;

END_FUNCTION

// mobject-converters/Converters/TIME_TO_/TryConvert_TIME_TO_DWORD
FUNCTION TryConvert_TIME_TO_DWORD : BOOL
VAR_INPUT
	in : TIME;
	out : REFERENCE TO DWORD;
END_VAR

out := TIME_TO_DWORD(in);
TryConvert_TIME_TO_DWORD := TRUE;

END_FUNCTION

// mobject-converters/Converters/TIME_TO_/TryConvert_TIME_TO_LWORD
FUNCTION TryConvert_TIME_TO_LWORD : BOOL
VAR_INPUT
	in : TIME;
	out : REFERENCE TO LWORD;
END_VAR

out := TIME_TO_LWORD(in);
TryConvert_TIME_TO_LWORD := TRUE;

END_FUNCTION

// mobject-converters/Converters/TIME_TO_/TryConvert_TIME_TO_SINT
FUNCTION TryConvert_TIME_TO_SINT : BOOL
VAR_INPUT
	in : TIME;
	out : REFERENCE TO SINT;
END_VAR

IF in > DatatypeLimits.MAX_VALUE_OF_TIME_WHICH_CAN_BE_HELD_IN_A_SINT THEN
	RETURN;
END_IF

out := TIME_TO_SINT(in);
TryConvert_TIME_TO_SINT := TRUE;

END_FUNCTION

// mobject-converters/Converters/TIME_TO_/TryConvert_TIME_TO_INT
FUNCTION TryConvert_TIME_TO_INT : BOOL
VAR_INPUT
	in : TIME;
	out : REFERENCE TO INT;
END_VAR

IF in > DatatypeLimits.MAX_VALUE_OF_TIME_WHICH_CAN_BE_HELD_IN_A_INT THEN
	RETURN;
END_IF

out := TIME_TO_INT(in);
TryConvert_TIME_TO_INT := TRUE;

END_FUNCTION

// mobject-converters/Converters/TIME_TO_/TryConvert_TIME_TO_DINT
FUNCTION TryConvert_TIME_TO_DINT : BOOL
VAR_INPUT
	in : TIME;
	out : REFERENCE TO DINT;
END_VAR

IF in > DatatypeLimits.MAX_VALUE_OF_TIME_WHICH_CAN_BE_HELD_IN_A_DINT THEN
	RETURN;
END_IF

out := TIME_TO_DINT(in);
TryConvert_TIME_TO_DINT := TRUE;

END_FUNCTION

// mobject-converters/Converters/TIME_TO_/TryConvert_TIME_TO_LINT
FUNCTION TryConvert_TIME_TO_LINT : BOOL
VAR_INPUT
	in : TIME;
	out : REFERENCE TO LINT;
END_VAR

out := TIME_TO_LINT(in);
TryConvert_TIME_TO_LINT := TRUE;

END_FUNCTION

// mobject-converters/Converters/TIME_TO_/TryConvert_TIME_TO_USINT
FUNCTION TryConvert_TIME_TO_USINT : BOOL
VAR_INPUT
	in : TIME;
	out : REFERENCE TO USINT;
END_VAR

IF in > DatatypeLimits.MAX_VALUE_OF_TIME_WHICH_CAN_BE_HELD_IN_A_USINT THEN
	RETURN;
END_IF

out := TIME_TO_USINT(in);
TryConvert_TIME_TO_USINT := TRUE;

END_FUNCTION

// mobject-converters/Converters/TIME_TO_/TryConvert_TIME_TO_UINT
FUNCTION TryConvert_TIME_TO_UINT : BOOL
VAR_INPUT
	in : TIME;
	out : REFERENCE TO UINT;
END_VAR

IF in > DatatypeLimits.MAX_VALUE_OF_TIME_WHICH_CAN_BE_HELD_IN_A_UINT THEN
	RETURN;
END_IF

out := TIME_TO_UINT(in);
TryConvert_TIME_TO_UINT := TRUE;

END_FUNCTION

// mobject-converters/Converters/TIME_TO_/TryConvert_TIME_TO_UDINT
FUNCTION TryConvert_TIME_TO_UDINT : BOOL
VAR_INPUT
	in : TIME;
	out : REFERENCE TO UDINT;
END_VAR

out := TIME_TO_UDINT(in);
TryConvert_TIME_TO_UDINT := TRUE;

END_FUNCTION

// mobject-converters/Converters/TIME_TO_/TryConvert_TIME_TO_ULINT
FUNCTION TryConvert_TIME_TO_ULINT : BOOL
VAR_INPUT
	in : TIME;
	out : REFERENCE TO ULINT;
END_VAR

out := TIME_TO_ULINT(in);
TryConvert_TIME_TO_ULINT := TRUE;

END_FUNCTION

// mobject-converters/Converters/TIME_TO_/TryConvert_TIME_TO_REAL
FUNCTION TryConvert_TIME_TO_REAL : BOOL
VAR_INPUT
	in : TIME;
	out : REFERENCE TO REAL;
END_VAR

out := TIME_TO_REAL(in);
TryConvert_TIME_TO_REAL := TRUE;

END_FUNCTION

// mobject-converters/Converters/TIME_TO_/TryConvert_TIME_TO_LREAL
FUNCTION TryConvert_TIME_TO_LREAL : BOOL
VAR_INPUT
	in : TIME;
	out : REFERENCE TO LREAL;
END_VAR

out := TIME_TO_LREAL(in);
TryConvert_TIME_TO_LREAL := TRUE;

END_FUNCTION

// mobject-converters/Converters/TIME_TO_/TryConvert_TIME_TO_TIME
FUNCTION TryConvert_TIME_TO_TIME : BOOL
VAR_INPUT
	in : TIME;
	out : REFERENCE TO TIME;
END_VAR

out := in;
TryConvert_TIME_TO_TIME := TRUE;

END_FUNCTION

// mobject-converters/Converters/TIME_TO_/TryConvert_TIME_TO_TOD
FUNCTION TryConvert_TIME_TO_TOD : BOOL
VAR_INPUT
	in : TIME;
	out : REFERENCE TO TOD;
END_VAR

IF in > DatatypeLimits.MAX_VALUE_OF_TIME_WHICH_CAN_BE_HELD_IN_A_TOD THEN
	RETURN;
END_IF

out := TIME_TO_TOD(in);
TryConvert_TIME_TO_TOD := TRUE;

END_FUNCTION

// mobject-converters/Converters/TIME_TO_/TryConvert_TIME_TO_DT
FUNCTION TryConvert_TIME_TO_DT : BOOL
VAR_INPUT
	in : TIME;
	out : REFERENCE TO DT;
END_VAR

out := TIME_TO_DT(in);
TryConvert_TIME_TO_DT := TRUE;

END_FUNCTION

// mobject-converters/Converters/TIME_TO_/TryConvert_TIME_TO_STRING
FUNCTION TryConvert_TIME_TO_STRING : BOOL
VAR_INPUT
	in : TIME;
	out : REFERENCE TO STRING;
END_VAR

out := TIME_TO_STRING(in);
TryConvert_TIME_TO_STRING := TRUE;

END_FUNCTION

// mobject-converters/Converters/TOD_TO_/TryConvert_TOD_TO_BOOL
FUNCTION TryConvert_TOD_TO_BOOL : BOOL
VAR_INPUT
	in : TOD;
	out : REFERENCE TO BOOL;
END_VAR

out := TOD_TO_BOOL(in);
TryConvert_TOD_TO_BOOL := TRUE;

END_FUNCTION

// mobject-converters/Converters/TOD_TO_/TryConvert_TOD_TO_BYTE
FUNCTION TryConvert_TOD_TO_BYTE : BOOL
VAR_INPUT
	in : TOD;
	out : REFERENCE TO BYTE;
END_VAR

IF in > DatatypeLimits.MAX_VALUE_OF_TOD_WHICH_CAN_BE_HELD_IN_A_BYTE THEN
	RETURN;
END_IF

out := TOD_TO_BYTE(in);
TryConvert_TOD_TO_BYTE := TRUE;

END_FUNCTION

// mobject-converters/Converters/TOD_TO_/TryConvert_TOD_TO_DATE
FUNCTION TryConvert_TOD_TO_DATE : BOOL
VAR_INPUT
	in : TOD;
	out : REFERENCE TO DATE;
END_VAR

out := TOD_TO_DATE(in);
TryConvert_TOD_TO_DATE := TRUE;

END_FUNCTION

// mobject-converters/Converters/TOD_TO_/TryConvert_TOD_TO_Destination
FUNCTION TryConvert_TOD_TO_Destination : BOOL
VAR_INPUT
	in : TOD;
	out : ANY;
END_VAR
VAR
	convertResult : BOOL := FALSE;
	convertAddress : PVOID;
	_BOOL : BOOL;
	_BYTE : BYTE;
	_WORD : WORD;
	_DWORD : DWORD;
	_LWORD : LWORD;
	_SINT : SINT;
	_INT : INT;
	_DINT : DINT;
	_LINT : LINT;
	_USINT : USINT;
	_UINT : UINT;
	_UDINT : UDINT;
	_ULINT : ULINT;
	_REAL : REAL;
	_LREAL : LREAL;
	_TIME : TIME;
	_TOD : TOD;
	_DATE : DATE;
	_DT : DT;
	_STRING : STRING;
END_VAR

CASE out.TypeClass OF
	__SYSTEM.TYPE_CLASS.TYPE_BOOL:
	
	convertResult := TryConvert_TOD_TO_BOOL(in, _BOOL);
	IF convertResult THEN
		convertAddress := ADR(_BOOL);
	END_IF
	
	__SYSTEM.TYPE_CLASS.TYPE_BYTE:
	
	convertResult := TryConvert_TOD_TO_BYTE(in, _BYTE);
	IF convertResult THEN
		convertAddress := ADR(_BYTE);
	END_IF
	
	__SYSTEM.TYPE_CLASS.TYPE_WORD:
	
	convertResult := TryConvert_TOD_TO_WORD(in, _WORD);
	IF convertResult THEN
		convertAddress := ADR(_WORD);
	END_IF
	
	__SYSTEM.TYPE_CLASS.TYPE_DWORD:
	
	convertResult := TryConvert_TOD_TO_DWORD(in, _DWORD);
	IF convertResult THEN
		convertAddress := ADR(_DWORD);
	END_IF
	
	__SYSTEM.TYPE_CLASS.TYPE_LWORD:
	
	convertResult := TryConvert_TOD_TO_LWORD(in, _LWORD);
	IF convertResult THEN
		convertAddress := ADR(_LWORD);
	END_IF
	
	__SYSTEM.TYPE_CLASS.TYPE_SINT:
	
	convertResult := TryConvert_TOD_TO_SINT(in, _SINT);
	IF convertResult THEN
		convertAddress := ADR(_SINT);
	END_IF
	
	__SYSTEM.TYPE_CLASS.TYPE_INT:
	
	convertResult := TryConvert_TOD_TO_INT(in, _INT);
	IF convertResult THEN
		convertAddress := ADR(_INT);
	END_IF
	
	__SYSTEM.TYPE_CLASS.TYPE_DINT:
	
	convertResult := TryConvert_TOD_TO_DINT(in, _DINT);
	IF convertResult THEN
		convertAddress := ADR(_DINT);
	END_IF
	
	__SYSTEM.TYPE_CLASS.TYPE_LINT:
	
	convertResult := TryConvert_TOD_TO_LINT(in, _LINT);
	IF convertResult THEN
		convertAddress := ADR(_LINT);
	END_IF
	
	__SYSTEM.TYPE_CLASS.TYPE_USINT:
	
	convertResult := TryConvert_TOD_TO_USINT(in, _USINT);
	IF convertResult THEN
		convertAddress := ADR(_USINT);
	END_IF
	
	__SYSTEM.TYPE_CLASS.TYPE_UINT:
	
	convertResult := TryConvert_TOD_TO_UINT(in, _UINT);
	IF convertResult THEN
		convertAddress := ADR(_UINT);
	END_IF
	
	__SYSTEM.TYPE_CLASS.TYPE_UDINT:
	
	convertResult := TryConvert_TOD_TO_UDINT(in, _UDINT);
	IF convertResult THEN
		convertAddress := ADR(_UDINT);
	END_IF
	
	__SYSTEM.TYPE_CLASS.TYPE_ULINT:
	
	convertResult := TryConvert_TOD_TO_ULINT(in, _ULINT);
	IF convertResult THEN
		convertAddress := ADR(_ULINT);
	END_IF
	
	__SYSTEM.TYPE_CLASS.TYPE_REAL:
	
	convertResult := TryConvert_TOD_TO_REAL(in, _REAL);
	IF convertResult THEN
		convertAddress := ADR(_REAL);
	END_IF
	
	__SYSTEM.TYPE_CLASS.TYPE_LREAL:
	
	convertResult := TryConvert_TOD_TO_LREAL(in, _LREAL);
	IF convertResult THEN
		convertAddress := ADR(_LREAL);
	END_IF
	
	__SYSTEM.TYPE_CLASS.TYPE_TIME:
	
	convertResult := TryConvert_TOD_TO_TIME(in, _TIME);
	IF convertResult THEN
		convertAddress := ADR(_TIME);
	END_IF
	
	__SYSTEM.TYPE_CLASS.TYPE_TIMEOFDAY:
	
	convertResult := TryConvert_TOD_TO_TOD(in, _TOD);
	IF convertResult THEN
		convertAddress := ADR(_TOD);
	END_IF
	
	__SYSTEM.TYPE_CLASS.TYPE_DATE:
	
	convertResult := TryConvert_TOD_TO_DATE(in, _DATE);
	IF convertResult THEN
		convertAddress := ADR(_DATE);
	END_IF
	
	__SYSTEM.TYPE_CLASS.TYPE_DATEANDTIME:
	
	convertResult := TryConvert_TOD_TO_DT(in, _DT);
	IF convertResult THEN
		convertAddress := ADR(_DT);
	END_IF
	
	__SYSTEM.TYPE_CLASS.TYPE_STRING:
	
	convertResult := TryConvert_TOD_TO_STRING(in, _STRING);
	IF convertResult THEN
		convertAddress := ADR(_STRING);
	END_IF
	
END_CASE

IF convertResult THEN
	memcpy(out.pValue,convertAddress,DINT_TO_UDINT(out.diSize));
END_IF

TryConvert_TOD_TO_Destination := convertResult;

END_FUNCTION

// mobject-converters/Converters/TOD_TO_/TryConvert_TOD_TO_WORD
FUNCTION TryConvert_TOD_TO_WORD : BOOL
VAR_INPUT
	in : TOD;
	out : REFERENCE TO WORD;
END_VAR

IF in > DatatypeLimits.MAX_VALUE_OF_TOD_WHICH_CAN_BE_HELD_IN_A_WORD THEN
	RETURN;
END_IF

out := TOD_TO_WORD(in);
TryConvert_TOD_TO_WORD := TRUE;

END_FUNCTION

// mobject-converters/Converters/TOD_TO_/TryConvert_TOD_TO_DWORD
FUNCTION TryConvert_TOD_TO_DWORD : BOOL
VAR_INPUT
	in : TOD;
	out : REFERENCE TO DWORD;
END_VAR

out := TOD_TO_DWORD(in);
TryConvert_TOD_TO_DWORD := TRUE;

END_FUNCTION

// mobject-converters/Converters/TOD_TO_/TryConvert_TOD_TO_LWORD
FUNCTION TryConvert_TOD_TO_LWORD : BOOL
VAR_INPUT
	in : TOD;
	out : REFERENCE TO LWORD;
END_VAR

out := TOD_TO_LWORD(in);
TryConvert_TOD_TO_LWORD := TRUE;

END_FUNCTION

// mobject-converters/Converters/TOD_TO_/TryConvert_TOD_TO_SINT
FUNCTION TryConvert_TOD_TO_SINT : BOOL
VAR_INPUT
	in : TOD;
	out : REFERENCE TO SINT;
END_VAR

IF in > DatatypeLimits.MAX_VALUE_OF_TOD_WHICH_CAN_BE_HELD_IN_A_SINT THEN
	RETURN;
END_IF

out := TOD_TO_SINT(in);
TryConvert_TOD_TO_SINT := TRUE;

END_FUNCTION

// mobject-converters/Converters/TOD_TO_/TryConvert_TOD_TO_INT
FUNCTION TryConvert_TOD_TO_INT : BOOL
VAR_INPUT
	in : TOD;
	out : REFERENCE TO INT;
END_VAR

IF in > DatatypeLimits.MAX_VALUE_OF_TOD_WHICH_CAN_BE_HELD_IN_A_INT THEN
	RETURN;
END_IF

out := TOD_TO_INT(in);
TryConvert_TOD_TO_INT := TRUE;

END_FUNCTION

// mobject-converters/Converters/TOD_TO_/TryConvert_TOD_TO_DINT
FUNCTION TryConvert_TOD_TO_DINT : BOOL
VAR_INPUT
	in : TOD;
	out : REFERENCE TO DINT;
END_VAR

out := TOD_TO_DINT(in);
TryConvert_TOD_TO_DINT := TRUE;

END_FUNCTION

// mobject-converters/Converters/TOD_TO_/TryConvert_TOD_TO_LINT
FUNCTION TryConvert_TOD_TO_LINT : BOOL
VAR_INPUT
	in : TOD;
	out : REFERENCE TO LINT;
END_VAR

out := TOD_TO_LINT(in);
TryConvert_TOD_TO_LINT := TRUE;

END_FUNCTION

// mobject-converters/Converters/TOD_TO_/TryConvert_TOD_TO_USINT
FUNCTION TryConvert_TOD_TO_USINT : BOOL
VAR_INPUT
	in : TOD;
	out : REFERENCE TO USINT;
END_VAR

IF in > DatatypeLimits.MAX_VALUE_OF_TOD_WHICH_CAN_BE_HELD_IN_A_USINT THEN
	RETURN;
END_IF

out := TOD_TO_USINT(in);
TryConvert_TOD_TO_USINT := TRUE;

END_FUNCTION

// mobject-converters/Converters/TOD_TO_/TryConvert_TOD_TO_UINT
FUNCTION TryConvert_TOD_TO_UINT : BOOL
VAR_INPUT
	in : TOD;
	out : REFERENCE TO UINT;
END_VAR

IF in > DatatypeLimits.MAX_VALUE_OF_TOD_WHICH_CAN_BE_HELD_IN_A_UINT THEN
	RETURN;
END_IF

out := TOD_TO_UINT(in);
TryConvert_TOD_TO_UINT := TRUE;

END_FUNCTION

// mobject-converters/Converters/TOD_TO_/TryConvert_TOD_TO_UDINT
FUNCTION TryConvert_TOD_TO_UDINT : BOOL
VAR_INPUT
	in : TOD;
	out : REFERENCE TO UDINT;
END_VAR

out := TOD_TO_UDINT(in);
TryConvert_TOD_TO_UDINT := TRUE;

END_FUNCTION

// mobject-converters/Converters/TOD_TO_/TryConvert_TOD_TO_ULINT
FUNCTION TryConvert_TOD_TO_ULINT : BOOL
VAR_INPUT
	in : TOD;
	out : REFERENCE TO ULINT;
END_VAR

out := TOD_TO_ULINT(in);
TryConvert_TOD_TO_ULINT := TRUE;

END_FUNCTION

// mobject-converters/Converters/TOD_TO_/TryConvert_TOD_TO_REAL
FUNCTION TryConvert_TOD_TO_REAL : BOOL
VAR_INPUT
	in : TOD;
	out : REFERENCE TO REAL;
END_VAR

out := TOD_TO_REAL(in);
TryConvert_TOD_TO_REAL := TRUE;

END_FUNCTION

// mobject-converters/Converters/TOD_TO_/TryConvert_TOD_TO_LREAL
FUNCTION TryConvert_TOD_TO_LREAL : BOOL
VAR_INPUT
	in : TOD;
	out : REFERENCE TO LREAL;
END_VAR

out := TOD_TO_LREAL(in);
TryConvert_TOD_TO_LREAL := TRUE;

END_FUNCTION

// mobject-converters/Converters/TOD_TO_/TryConvert_TOD_TO_TIME
FUNCTION TryConvert_TOD_TO_TIME : BOOL
VAR_INPUT
	in : TOD;
	out : REFERENCE TO TIME;
END_VAR

out := TOD_TO_TIME(in);
TryConvert_TOD_TO_TIME := TRUE;

END_FUNCTION

// mobject-converters/Converters/TOD_TO_/TryConvert_TOD_TO_TOD
FUNCTION TryConvert_TOD_TO_TOD : BOOL
VAR_INPUT
	in : TOD;
	out : REFERENCE TO TOD;
END_VAR

out := in;
TryConvert_TOD_TO_TOD := TRUE;

END_FUNCTION

// mobject-converters/Converters/TOD_TO_/TryConvert_TOD_TO_DT
FUNCTION TryConvert_TOD_TO_DT : BOOL
VAR_INPUT
	in : TOD;
	out : REFERENCE TO DT;
END_VAR

out := TOD_TO_DT(in);
TryConvert_TOD_TO_DT := TRUE;

END_FUNCTION

// mobject-converters/Converters/TOD_TO_/TryConvert_TOD_TO_STRING
FUNCTION TryConvert_TOD_TO_STRING : BOOL
VAR_INPUT
	in : TOD;
	out : REFERENCE TO STRING;
END_VAR

out := TOD_TO_STRING(in);
TryConvert_TOD_TO_STRING := TRUE;

END_FUNCTION

// mobject-converters/Converters/UDINT_TO_/TryConvert_UDINT_TO_BOOL
FUNCTION TryConvert_UDINT_TO_BOOL : BOOL
VAR_INPUT
	in : UDINT;
	out : REFERENCE TO BOOL;
END_VAR

out := UDINT_TO_BOOL(in);
TryConvert_UDINT_TO_BOOL := TRUE;

END_FUNCTION

// mobject-converters/Converters/UDINT_TO_/TryConvert_UDINT_TO_BYTE
FUNCTION TryConvert_UDINT_TO_BYTE : BOOL
VAR_INPUT
	in : UDINT;
	out : REFERENCE TO BYTE;
END_VAR

IF in > DatatypeLimits.MAX_VALUE_OF_UDINT_WHICH_CAN_BE_HELD_IN_A_BYTE THEN
	RETURN;
END_IF

out := UDINT_TO_BYTE(in);
TryConvert_UDINT_TO_BYTE := TRUE;

END_FUNCTION

// mobject-converters/Converters/UDINT_TO_/TryConvert_UDINT_TO_DATE
FUNCTION TryConvert_UDINT_TO_DATE : BOOL
VAR_INPUT
	in : UDINT;
	out : REFERENCE TO DATE;
END_VAR

out := UDINT_TO_DATE(in);
TryConvert_UDINT_TO_DATE := TRUE;

END_FUNCTION

// mobject-converters/Converters/UDINT_TO_/TryConvert_UDINT_TO_Destination
FUNCTION TryConvert_UDINT_TO_Destination : BOOL
VAR_INPUT
	in : UDINT;
	out : ANY;
END_VAR
VAR
	convertResult : BOOL := FALSE;
	convertAddress : PVOID;
	_BOOL : BOOL;
	_BYTE : BYTE;
	_WORD : WORD;
	_DWORD : DWORD;
	_LWORD : LWORD;
	_SINT : SINT;
	_INT : INT;
	_DINT : DINT;
	_LINT : LINT;
	_USINT : USINT;
	_UINT : UINT;
	_UDINT : UDINT;
	_ULINT : ULINT;
	_REAL : REAL;
	_LREAL : LREAL;
	_TIME : TIME;
	_TOD : TOD;
	_DATE : DATE;
	_DT : DT;
	_STRING : STRING;
END_VAR

CASE out.TypeClass OF
	__SYSTEM.TYPE_CLASS.TYPE_BOOL:
	
	convertResult := TryConvert_UDINT_TO_BOOL(in, _BOOL);
	IF convertResult THEN
		convertAddress := ADR(_BOOL);
	END_IF
	
	__SYSTEM.TYPE_CLASS.TYPE_BYTE:
	
	convertResult := TryConvert_UDINT_TO_BYTE(in, _BYTE);
	IF convertResult THEN
		convertAddress := ADR(_BYTE);
	END_IF
	
	__SYSTEM.TYPE_CLASS.TYPE_WORD:
	
	convertResult := TryConvert_UDINT_TO_WORD(in, _WORD);
	IF convertResult THEN
		convertAddress := ADR(_WORD);
	END_IF
	
	__SYSTEM.TYPE_CLASS.TYPE_DWORD:
	
	convertResult := TryConvert_UDINT_TO_DWORD(in, _DWORD);
	IF convertResult THEN
		convertAddress := ADR(_DWORD);
	END_IF
	
	__SYSTEM.TYPE_CLASS.TYPE_LWORD:
	
	convertResult := TryConvert_UDINT_TO_LWORD(in, _LWORD);
	IF convertResult THEN
		convertAddress := ADR(_LWORD);
	END_IF
	
	__SYSTEM.TYPE_CLASS.TYPE_SINT:
	
	convertResult := TryConvert_UDINT_TO_SINT(in, _SINT);
	IF convertResult THEN
		convertAddress := ADR(_SINT);
	END_IF
	
	__SYSTEM.TYPE_CLASS.TYPE_INT:
	
	convertResult := TryConvert_UDINT_TO_INT(in, _INT);
	IF convertResult THEN
		convertAddress := ADR(_INT);
	END_IF
	
	__SYSTEM.TYPE_CLASS.TYPE_DINT:
	
	convertResult := TryConvert_UDINT_TO_DINT(in, _DINT);
	IF convertResult THEN
		convertAddress := ADR(_DINT);
	END_IF
	
	__SYSTEM.TYPE_CLASS.TYPE_LINT:
	
	convertResult := TryConvert_UDINT_TO_LINT(in, _LINT);
	IF convertResult THEN
		convertAddress := ADR(_LINT);
	END_IF
	
	__SYSTEM.TYPE_CLASS.TYPE_USINT:
	
	convertResult := TryConvert_UDINT_TO_USINT(in, _USINT);
	IF convertResult THEN
		convertAddress := ADR(_USINT);
	END_IF
	
	__SYSTEM.TYPE_CLASS.TYPE_UINT:
	
	convertResult := TryConvert_UDINT_TO_UINT(in, _UINT);
	IF convertResult THEN
		convertAddress := ADR(_UINT);
	END_IF
	
	__SYSTEM.TYPE_CLASS.TYPE_UDINT:
	
	convertResult := TryConvert_UDINT_TO_UDINT(in, _UDINT);
	IF convertResult THEN
		convertAddress := ADR(_UDINT);
	END_IF
	
	__SYSTEM.TYPE_CLASS.TYPE_ULINT:
	
	convertResult := TryConvert_UDINT_TO_ULINT(in, _ULINT);
	IF convertResult THEN
		convertAddress := ADR(_ULINT);
	END_IF
	
	__SYSTEM.TYPE_CLASS.TYPE_REAL:
	
	convertResult := TryConvert_UDINT_TO_REAL(in, _REAL);
	IF convertResult THEN
		convertAddress := ADR(_REAL);
	END_IF
	
	__SYSTEM.TYPE_CLASS.TYPE_LREAL:
	
	convertResult := TryConvert_UDINT_TO_LREAL(in, _LREAL);
	IF convertResult THEN
		convertAddress := ADR(_LREAL);
	END_IF
	
	__SYSTEM.TYPE_CLASS.TYPE_TIME:
	
	convertResult := TryConvert_UDINT_TO_TIME(in, _TIME);
	IF convertResult THEN
		convertAddress := ADR(_TIME);
	END_IF
	
	__SYSTEM.TYPE_CLASS.TYPE_TIMEOFDAY:
	
	convertResult := TryConvert_UDINT_TO_TOD(in, _TOD);
	IF convertResult THEN
		convertAddress := ADR(_TOD);
	END_IF
	
	__SYSTEM.TYPE_CLASS.TYPE_DATE:
	
	convertResult := TryConvert_UDINT_TO_DATE(in, _DATE);
	IF convertResult THEN
		convertAddress := ADR(_DATE);
	END_IF
	
	__SYSTEM.TYPE_CLASS.TYPE_DATEANDTIME:
	
	convertResult := TryConvert_UDINT_TO_DT(in, _DT);
	IF convertResult THEN
		convertAddress := ADR(_DT);
	END_IF
	
	__SYSTEM.TYPE_CLASS.TYPE_STRING:
	
	convertResult := TryConvert_UDINT_TO_STRING(in, _STRING);
	IF convertResult THEN
		convertAddress := ADR(_STRING);
	END_IF
	
END_CASE

IF convertResult THEN
	memcpy(out.pValue,convertAddress,DINT_TO_UDINT(out.diSize));
END_IF

TryConvert_UDINT_TO_Destination := convertResult;

END_FUNCTION

// mobject-converters/Converters/UDINT_TO_/TryConvert_UDINT_TO_WORD
FUNCTION TryConvert_UDINT_TO_WORD : BOOL
VAR_INPUT
	in : UDINT;
	out : REFERENCE TO WORD;
END_VAR

IF in > DatatypeLimits.MAX_VALUE_OF_UDINT_WHICH_CAN_BE_HELD_IN_A_WORD THEN
	RETURN;
END_IF

out := UDINT_TO_WORD(in);
TryConvert_UDINT_TO_WORD := TRUE;

END_FUNCTION

// mobject-converters/Converters/UDINT_TO_/TryConvert_UDINT_TO_DWORD
FUNCTION TryConvert_UDINT_TO_DWORD : BOOL
VAR_INPUT
	in : UDINT;
	out : REFERENCE TO DWORD;
END_VAR

out := UDINT_TO_DWORD(in);
TryConvert_UDINT_TO_DWORD := TRUE;

END_FUNCTION

// mobject-converters/Converters/UDINT_TO_/TryConvert_UDINT_TO_LWORD
FUNCTION TryConvert_UDINT_TO_LWORD : BOOL
VAR_INPUT
	in : UDINT;
	out : REFERENCE TO LWORD;
END_VAR

out := UDINT_TO_LWORD(in);
TryConvert_UDINT_TO_LWORD := TRUE;

END_FUNCTION

// mobject-converters/Converters/UDINT_TO_/TryConvert_UDINT_TO_SINT
FUNCTION TryConvert_UDINT_TO_SINT : BOOL
VAR_INPUT
	in : UDINT;
	out : REFERENCE TO SINT;
END_VAR

IF in > DatatypeLimits.MAX_VALUE_OF_UDINT_WHICH_CAN_BE_HELD_IN_A_SINT THEN
	RETURN;
END_IF

out := UDINT_TO_SINT(in);
TryConvert_UDINT_TO_SINT := TRUE;

END_FUNCTION

// mobject-converters/Converters/UDINT_TO_/TryConvert_UDINT_TO_INT
FUNCTION TryConvert_UDINT_TO_INT : BOOL
VAR_INPUT
	in : UDINT;
	out : REFERENCE TO INT;
END_VAR

IF in > DatatypeLimits.MAX_VALUE_OF_UDINT_WHICH_CAN_BE_HELD_IN_A_INT THEN
	RETURN;
END_IF

out := UDINT_TO_INT(in);
TryConvert_UDINT_TO_INT := TRUE;

END_FUNCTION

// mobject-converters/Converters/UDINT_TO_/TryConvert_UDINT_TO_DINT
FUNCTION TryConvert_UDINT_TO_DINT : BOOL
VAR_INPUT
	in : UDINT;
	out : REFERENCE TO DINT;
END_VAR

IF in > DatatypeLimits.MAX_VALUE_OF_UDINT_WHICH_CAN_BE_HELD_IN_A_DINT THEN
	RETURN;
END_IF

out := UDINT_TO_DINT(in);
TryConvert_UDINT_TO_DINT := TRUE;

END_FUNCTION

// mobject-converters/Converters/UDINT_TO_/TryConvert_UDINT_TO_LINT
FUNCTION TryConvert_UDINT_TO_LINT : BOOL
VAR_INPUT
	in : UDINT;
	out : REFERENCE TO LINT;
END_VAR

out := UDINT_TO_LINT(in);
TryConvert_UDINT_TO_LINT := TRUE;

END_FUNCTION

// mobject-converters/Converters/UDINT_TO_/TryConvert_UDINT_TO_USINT
FUNCTION TryConvert_UDINT_TO_USINT : BOOL
VAR_INPUT
	in : UDINT;
	out : REFERENCE TO USINT;
END_VAR

IF in > DatatypeLimits.MAX_VALUE_OF_UDINT_WHICH_CAN_BE_HELD_IN_A_USINT THEN
	RETURN;
END_IF

out := UDINT_TO_USINT(in);
TryConvert_UDINT_TO_USINT := TRUE;

END_FUNCTION

// mobject-converters/Converters/UDINT_TO_/TryConvert_UDINT_TO_UINT
FUNCTION TryConvert_UDINT_TO_UINT : BOOL
VAR_INPUT
	in : UDINT;
	out : REFERENCE TO UINT;
END_VAR

IF in > DatatypeLimits.MAX_VALUE_OF_UDINT_WHICH_CAN_BE_HELD_IN_A_UINT THEN
	RETURN;
END_IF

out := UDINT_TO_UINT(in);
TryConvert_UDINT_TO_UINT := TRUE;

END_FUNCTION

// mobject-converters/Converters/UDINT_TO_/TryConvert_UDINT_TO_UDINT
FUNCTION TryConvert_UDINT_TO_UDINT : BOOL
VAR_INPUT
	in : UDINT;
	out : REFERENCE TO UDINT;
END_VAR

out := in;
TryConvert_UDINT_TO_UDINT := TRUE;

END_FUNCTION

// mobject-converters/Converters/UDINT_TO_/TryConvert_UDINT_TO_ULINT
FUNCTION TryConvert_UDINT_TO_ULINT : BOOL
VAR_INPUT
	in : UDINT;
	out : REFERENCE TO ULINT;
END_VAR

out := UDINT_TO_ULINT(in);
TryConvert_UDINT_TO_ULINT := TRUE;

END_FUNCTION

// mobject-converters/Converters/UDINT_TO_/TryConvert_UDINT_TO_REAL
FUNCTION TryConvert_UDINT_TO_REAL : BOOL
VAR_INPUT
	in : UDINT;
	out : REFERENCE TO REAL;
END_VAR

out := UDINT_TO_REAL(in);
TryConvert_UDINT_TO_REAL := TRUE;

END_FUNCTION

// mobject-converters/Converters/UDINT_TO_/TryConvert_UDINT_TO_LREAL
FUNCTION TryConvert_UDINT_TO_LREAL : BOOL
VAR_INPUT
	in : UDINT;
	out : REFERENCE TO LREAL;
END_VAR

out := UDINT_TO_LREAL(in);
TryConvert_UDINT_TO_LREAL := TRUE;

END_FUNCTION

// mobject-converters/Converters/UDINT_TO_/TryConvert_UDINT_TO_TIME
FUNCTION TryConvert_UDINT_TO_TIME : BOOL
VAR_INPUT
	in : UDINT;
	out : REFERENCE TO TIME;
END_VAR

out := UDINT_TO_TIME(in);
TryConvert_UDINT_TO_TIME := TRUE;

END_FUNCTION

// mobject-converters/Converters/UDINT_TO_/TryConvert_UDINT_TO_TOD
FUNCTION TryConvert_UDINT_TO_TOD : BOOL
VAR_INPUT
	in : UDINT;
	out : REFERENCE TO TOD;
END_VAR

IF in > DatatypeLimits.MAX_VALUE_OF_UDINT_WHICH_CAN_BE_HELD_IN_A_TOD THEN
	RETURN;
END_IF

out := UDINT_TO_TOD(in);
TryConvert_UDINT_TO_TOD := TRUE;

END_FUNCTION

// mobject-converters/Converters/UDINT_TO_/TryConvert_UDINT_TO_DT
FUNCTION TryConvert_UDINT_TO_DT : BOOL
VAR_INPUT
	in : UDINT;
	out : REFERENCE TO DT;
END_VAR

out := UDINT_TO_DT(in);
TryConvert_UDINT_TO_DT := TRUE;

END_FUNCTION

// mobject-converters/Converters/UDINT_TO_/TryConvert_UDINT_TO_STRING
FUNCTION TryConvert_UDINT_TO_STRING : BOOL
VAR_INPUT
	in : UDINT;
	out : REFERENCE TO STRING;
END_VAR

out := UDINT_TO_STRING(in);
TryConvert_UDINT_TO_STRING := TRUE;

END_FUNCTION

// mobject-converters/Converters/UINT_TO_/TryConvert_UINT_TO_BOOL
FUNCTION TryConvert_UINT_TO_BOOL : BOOL
VAR_INPUT
	in : UINT;
	out : REFERENCE TO BOOL;
END_VAR

out := UINT_TO_BOOL(in);
TryConvert_UINT_TO_BOOL := TRUE;

END_FUNCTION

// mobject-converters/Converters/UINT_TO_/TryConvert_UINT_TO_BYTE
FUNCTION TryConvert_UINT_TO_BYTE : BOOL
VAR_INPUT
	in : UINT;
	out : REFERENCE TO BYTE;
END_VAR

IF in > DatatypeLimits.MAX_VALUE_OF_UINT_WHICH_CAN_BE_HELD_IN_A_BYTE THEN
	RETURN;
END_IF

out := UINT_TO_BYTE(in);
TryConvert_UINT_TO_BYTE := TRUE;

END_FUNCTION

// mobject-converters/Converters/UINT_TO_/TryConvert_UINT_TO_DATE
FUNCTION TryConvert_UINT_TO_DATE : BOOL
VAR_INPUT
	in : UINT;
	out : REFERENCE TO DATE;
END_VAR

out := UINT_TO_DATE(in);
TryConvert_UINT_TO_DATE := TRUE;

END_FUNCTION

// mobject-converters/Converters/UINT_TO_/TryConvert_UINT_TO_Destination
FUNCTION TryConvert_UINT_TO_Destination : BOOL
VAR_INPUT
	in : UINT;
	out : ANY;
END_VAR
VAR
	convertResult : BOOL := FALSE;
	convertAddress : PVOID;
	_BOOL : BOOL;
	_BYTE : BYTE;
	_WORD : WORD;
	_DWORD : DWORD;
	_LWORD : LWORD;
	_SINT : SINT;
	_INT : INT;
	_DINT : DINT;
	_LINT : LINT;
	_USINT : USINT;
	_UINT : UINT;
	_UDINT : UDINT;
	_ULINT : ULINT;
	_REAL : REAL;
	_LREAL : LREAL;
	_TIME : TIME;
	_TOD : TOD;
	_DATE : DATE;
	_DT : DT;
	_STRING : STRING;
END_VAR

CASE out.TypeClass OF
	__SYSTEM.TYPE_CLASS.TYPE_BOOL:
	
	convertResult := TryConvert_UINT_TO_BOOL(in, _BOOL);
	IF convertResult THEN
		convertAddress := ADR(_BOOL);
	END_IF
	
	__SYSTEM.TYPE_CLASS.TYPE_BYTE:
	
	convertResult := TryConvert_UINT_TO_BYTE(in, _BYTE);
	IF convertResult THEN
		convertAddress := ADR(_BYTE);
	END_IF
	
	__SYSTEM.TYPE_CLASS.TYPE_WORD:
	
	convertResult := TryConvert_UINT_TO_WORD(in, _WORD);
	IF convertResult THEN
		convertAddress := ADR(_WORD);
	END_IF
	
	__SYSTEM.TYPE_CLASS.TYPE_DWORD:
	
	convertResult := TryConvert_UINT_TO_DWORD(in, _DWORD);
	IF convertResult THEN
		convertAddress := ADR(_DWORD);
	END_IF
	
	__SYSTEM.TYPE_CLASS.TYPE_LWORD:
	
	convertResult := TryConvert_UINT_TO_LWORD(in, _LWORD);
	IF convertResult THEN
		convertAddress := ADR(_LWORD);
	END_IF
	
	__SYSTEM.TYPE_CLASS.TYPE_SINT:
	
	convertResult := TryConvert_UINT_TO_SINT(in, _SINT);
	IF convertResult THEN
		convertAddress := ADR(_SINT);
	END_IF
	
	__SYSTEM.TYPE_CLASS.TYPE_INT:
	
	convertResult := TryConvert_UINT_TO_INT(in, _INT);
	IF convertResult THEN
		convertAddress := ADR(_INT);
	END_IF
	
	__SYSTEM.TYPE_CLASS.TYPE_DINT:
	
	convertResult := TryConvert_UINT_TO_DINT(in, _DINT);
	IF convertResult THEN
		convertAddress := ADR(_DINT);
	END_IF
	
	__SYSTEM.TYPE_CLASS.TYPE_LINT:
	
	convertResult := TryConvert_UINT_TO_LINT(in, _LINT);
	IF convertResult THEN
		convertAddress := ADR(_LINT);
	END_IF
	
	__SYSTEM.TYPE_CLASS.TYPE_USINT:
	
	convertResult := TryConvert_UINT_TO_USINT(in, _USINT);
	IF convertResult THEN
		convertAddress := ADR(_USINT);
	END_IF
	
	__SYSTEM.TYPE_CLASS.TYPE_UINT:
	
	convertResult := TryConvert_UINT_TO_UINT(in, _UINT);
	IF convertResult THEN
		convertAddress := ADR(_UINT);
	END_IF
	
	__SYSTEM.TYPE_CLASS.TYPE_UDINT:
	
	convertResult := TryConvert_UINT_TO_UDINT(in, _UDINT);
	IF convertResult THEN
		convertAddress := ADR(_UDINT);
	END_IF
	
	__SYSTEM.TYPE_CLASS.TYPE_ULINT:
	
	convertResult := TryConvert_UINT_TO_ULINT(in, _ULINT);
	IF convertResult THEN
		convertAddress := ADR(_ULINT);
	END_IF
	
	__SYSTEM.TYPE_CLASS.TYPE_REAL:
	
	convertResult := TryConvert_UINT_TO_REAL(in, _REAL);
	IF convertResult THEN
		convertAddress := ADR(_REAL);
	END_IF
	
	__SYSTEM.TYPE_CLASS.TYPE_LREAL:
	
	convertResult := TryConvert_UINT_TO_LREAL(in, _LREAL);
	IF convertResult THEN
		convertAddress := ADR(_LREAL);
	END_IF
	
	__SYSTEM.TYPE_CLASS.TYPE_TIME:
	
	convertResult := TryConvert_UINT_TO_TIME(in, _TIME);
	IF convertResult THEN
		convertAddress := ADR(_TIME);
	END_IF
	
	__SYSTEM.TYPE_CLASS.TYPE_TIMEOFDAY:
	
	convertResult := TryConvert_UINT_TO_TOD(in, _TOD);
	IF convertResult THEN
		convertAddress := ADR(_TOD);
	END_IF
	
	__SYSTEM.TYPE_CLASS.TYPE_DATE:
	
	convertResult := TryConvert_UINT_TO_DATE(in, _DATE);
	IF convertResult THEN
		convertAddress := ADR(_DATE);
	END_IF
	
	__SYSTEM.TYPE_CLASS.TYPE_DATEANDTIME:
	
	convertResult := TryConvert_UINT_TO_DT(in, _DT);
	IF convertResult THEN
		convertAddress := ADR(_DT);
	END_IF
	
	__SYSTEM.TYPE_CLASS.TYPE_STRING:
	
	convertResult := TryConvert_UINT_TO_STRING(in, _STRING);
	IF convertResult THEN
		convertAddress := ADR(_STRING);
	END_IF
	
END_CASE

IF convertResult THEN
	memcpy(out.pValue,convertAddress,DINT_TO_UDINT(out.diSize));
END_IF

TryConvert_UINT_TO_Destination := convertResult;

END_FUNCTION

// mobject-converters/Converters/UINT_TO_/TryConvert_UINT_TO_WORD
FUNCTION TryConvert_UINT_TO_WORD : BOOL
VAR_INPUT
	in : UINT;
	out : REFERENCE TO WORD;
END_VAR

out := UINT_TO_WORD(in);
TryConvert_UINT_TO_WORD := TRUE;

END_FUNCTION

// mobject-converters/Converters/UINT_TO_/TryConvert_UINT_TO_DWORD
FUNCTION TryConvert_UINT_TO_DWORD : BOOL
VAR_INPUT
	in : UINT;
	out : REFERENCE TO DWORD;
END_VAR

out := UINT_TO_DWORD(in);
TryConvert_UINT_TO_DWORD := TRUE;

END_FUNCTION

// mobject-converters/Converters/UINT_TO_/TryConvert_UINT_TO_LWORD
FUNCTION TryConvert_UINT_TO_LWORD : BOOL
VAR_INPUT
	in : UINT;
	out : REFERENCE TO LWORD;
END_VAR

out := UINT_TO_LWORD(in);
TryConvert_UINT_TO_LWORD := TRUE;

END_FUNCTION

// mobject-converters/Converters/UINT_TO_/TryConvert_UINT_TO_SINT
FUNCTION TryConvert_UINT_TO_SINT : BOOL
VAR_INPUT
	in : UINT;
	out : REFERENCE TO SINT;
END_VAR

IF in > DatatypeLimits.MAX_VALUE_OF_UINT_WHICH_CAN_BE_HELD_IN_A_SINT THEN
	RETURN;
END_IF

out := UINT_TO_SINT(in);
TryConvert_UINT_TO_SINT := TRUE;

END_FUNCTION

// mobject-converters/Converters/UINT_TO_/TryConvert_UINT_TO_INT
FUNCTION TryConvert_UINT_TO_INT : BOOL
VAR_INPUT
	in : UINT;
	out : REFERENCE TO INT;
END_VAR

IF in > DatatypeLimits.MAX_VALUE_OF_UINT_WHICH_CAN_BE_HELD_IN_A_INT THEN
	RETURN;
END_IF

out := UINT_TO_INT(in);
TryConvert_UINT_TO_INT := TRUE;

END_FUNCTION

// mobject-converters/Converters/UINT_TO_/TryConvert_UINT_TO_DINT
FUNCTION TryConvert_UINT_TO_DINT : BOOL
VAR_INPUT
	in : UINT;
	out : REFERENCE TO DINT;
END_VAR

out := UINT_TO_DINT(in);
TryConvert_UINT_TO_DINT := TRUE;

END_FUNCTION

// mobject-converters/Converters/UINT_TO_/TryConvert_UINT_TO_LINT
FUNCTION TryConvert_UINT_TO_LINT : BOOL
VAR_INPUT
	in : UINT;
	out : REFERENCE TO LINT;
END_VAR

out := UINT_TO_LINT(in);
TryConvert_UINT_TO_LINT := TRUE;

END_FUNCTION

// mobject-converters/Converters/UINT_TO_/TryConvert_UINT_TO_USINT
FUNCTION TryConvert_UINT_TO_USINT : BOOL
VAR_INPUT
	in : UINT;
	out : REFERENCE TO USINT;
END_VAR

IF in > DatatypeLimits.MAX_VALUE_OF_UINT_WHICH_CAN_BE_HELD_IN_A_USINT THEN
	RETURN;
END_IF

out := UINT_TO_USINT(in);
TryConvert_UINT_TO_USINT := TRUE;

END_FUNCTION

// mobject-converters/Converters/UINT_TO_/TryConvert_UINT_TO_UINT
FUNCTION TryConvert_UINT_TO_UINT : BOOL
VAR_INPUT
	in : UINT;
	out : REFERENCE TO UINT;
END_VAR

out := in;
TryConvert_UINT_TO_UINT := TRUE;

END_FUNCTION

// mobject-converters/Converters/UINT_TO_/TryConvert_UINT_TO_UDINT
FUNCTION TryConvert_UINT_TO_UDINT : BOOL
VAR_INPUT
	in : UINT;
	out : REFERENCE TO UDINT;
END_VAR

out := UINT_TO_UDINT(in);
TryConvert_UINT_TO_UDINT := TRUE;

END_FUNCTION

// mobject-converters/Converters/UINT_TO_/TryConvert_UINT_TO_ULINT
FUNCTION TryConvert_UINT_TO_ULINT : BOOL
VAR_INPUT
	in : UINT;
	out : REFERENCE TO ULINT;
END_VAR

out := UINT_TO_ULINT(in);
TryConvert_UINT_TO_ULINT := TRUE;

END_FUNCTION

// mobject-converters/Converters/UINT_TO_/TryConvert_UINT_TO_REAL
FUNCTION TryConvert_UINT_TO_REAL : BOOL
VAR_INPUT
	in : UINT;
	out : REFERENCE TO REAL;
END_VAR

out := UINT_TO_REAL(in);
TryConvert_UINT_TO_REAL := TRUE;

END_FUNCTION

// mobject-converters/Converters/UINT_TO_/TryConvert_UINT_TO_LREAL
FUNCTION TryConvert_UINT_TO_LREAL : BOOL
VAR_INPUT
	in : UINT;
	out : REFERENCE TO LREAL;
END_VAR

out := UINT_TO_LREAL(in);
TryConvert_UINT_TO_LREAL := TRUE;

END_FUNCTION

// mobject-converters/Converters/UINT_TO_/TryConvert_UINT_TO_TIME
FUNCTION TryConvert_UINT_TO_TIME : BOOL
VAR_INPUT
	in : UINT;
	out : REFERENCE TO TIME;
END_VAR

out := UINT_TO_TIME(in);
TryConvert_UINT_TO_TIME := TRUE;

END_FUNCTION

// mobject-converters/Converters/UINT_TO_/TryConvert_UINT_TO_TOD
FUNCTION TryConvert_UINT_TO_TOD : BOOL
VAR_INPUT
	in : UINT;
	out : REFERENCE TO TOD;
END_VAR

out := UINT_TO_TOD(in);
TryConvert_UINT_TO_TOD := TRUE;

END_FUNCTION

// mobject-converters/Converters/UINT_TO_/TryConvert_UINT_TO_DT
FUNCTION TryConvert_UINT_TO_DT : BOOL
VAR_INPUT
	in : UINT;
	out : REFERENCE TO DT;
END_VAR

out := UINT_TO_DT(in);
TryConvert_UINT_TO_DT := TRUE;

END_FUNCTION

// mobject-converters/Converters/UINT_TO_/TryConvert_UINT_TO_STRING
FUNCTION TryConvert_UINT_TO_STRING : BOOL
VAR_INPUT
	in : UINT;
	out : REFERENCE TO STRING;
END_VAR

out := UINT_TO_STRING(in);
TryConvert_UINT_TO_STRING := TRUE;

END_FUNCTION

// mobject-converters/Converters/ULINT_TO_/TryConvert_ULINT_TO_BOOL
FUNCTION TryConvert_ULINT_TO_BOOL : BOOL
VAR_INPUT
	in : ULINT;
	out : REFERENCE TO BOOL;
END_VAR

out := ULINT_TO_BOOL(in);
TryConvert_ULINT_TO_BOOL := TRUE;

END_FUNCTION

// mobject-converters/Converters/ULINT_TO_/TryConvert_ULINT_TO_BYTE
FUNCTION TryConvert_ULINT_TO_BYTE : BOOL
VAR_INPUT
	in : ULINT;
	out : REFERENCE TO BYTE;
END_VAR

IF in > DatatypeLimits.MAX_VALUE_OF_ULINT_WHICH_CAN_BE_HELD_IN_A_BYTE THEN
	RETURN;
END_IF

out := ULINT_TO_BYTE(in);
TryConvert_ULINT_TO_BYTE := TRUE;

END_FUNCTION

// mobject-converters/Converters/ULINT_TO_/TryConvert_ULINT_TO_DATE
FUNCTION TryConvert_ULINT_TO_DATE : BOOL
VAR_INPUT
	in : ULINT;
	out : REFERENCE TO DATE;
END_VAR

IF in > DatatypeLimits.MAX_VALUE_OF_ULINT_WHICH_CAN_BE_HELD_IN_A_DATE THEN
	RETURN;
END_IF

out := ULINT_TO_DATE(in);
TryConvert_ULINT_TO_DATE := TRUE;

END_FUNCTION

// mobject-converters/Converters/ULINT_TO_/TryConvert_ULINT_TO_Destination
FUNCTION TryConvert_ULINT_TO_Destination : BOOL
VAR_INPUT
	in : ULINT;
	out : ANY;
END_VAR
VAR
	convertResult : BOOL := FALSE;
	convertAddress : PVOID;
	_BOOL : BOOL;
	_BYTE : BYTE;
	_WORD : WORD;
	_DWORD : DWORD;
	_LWORD : LWORD;
	_SINT : SINT;
	_INT : INT;
	_DINT : DINT;
	_LINT : LINT;
	_USINT : USINT;
	_UINT : UINT;
	_UDINT : UDINT;
	_ULINT : ULINT;
	_REAL : REAL;
	_LREAL : LREAL;
	_TIME : TIME;
	_TOD : TOD;
	_DATE : DATE;
	_DT : DT;
	_STRING : STRING;
END_VAR

CASE out.TypeClass OF
	__SYSTEM.TYPE_CLASS.TYPE_BOOL:
	
	convertResult := TryConvert_ULINT_TO_BOOL(in, _BOOL);
	IF convertResult THEN
		convertAddress := ADR(_BOOL);
	END_IF
	
	__SYSTEM.TYPE_CLASS.TYPE_BYTE:
	
	convertResult := TryConvert_ULINT_TO_BYTE(in, _BYTE);
	IF convertResult THEN
		convertAddress := ADR(_BYTE);
	END_IF
	
	__SYSTEM.TYPE_CLASS.TYPE_WORD:
	
	convertResult := TryConvert_ULINT_TO_WORD(in, _WORD);
	IF convertResult THEN
		convertAddress := ADR(_WORD);
	END_IF
	
	__SYSTEM.TYPE_CLASS.TYPE_DWORD:
	
	convertResult := TryConvert_ULINT_TO_DWORD(in, _DWORD);
	IF convertResult THEN
		convertAddress := ADR(_DWORD);
	END_IF
	
	__SYSTEM.TYPE_CLASS.TYPE_LWORD:
	
	convertResult := TryConvert_ULINT_TO_LWORD(in, _LWORD);
	IF convertResult THEN
		convertAddress := ADR(_LWORD);
	END_IF
	
	__SYSTEM.TYPE_CLASS.TYPE_SINT:
	
	convertResult := TryConvert_ULINT_TO_SINT(in, _SINT);
	IF convertResult THEN
		convertAddress := ADR(_SINT);
	END_IF
	
	__SYSTEM.TYPE_CLASS.TYPE_INT:
	
	convertResult := TryConvert_ULINT_TO_INT(in, _INT);
	IF convertResult THEN
		convertAddress := ADR(_INT);
	END_IF
	
	__SYSTEM.TYPE_CLASS.TYPE_DINT:
	
	convertResult := TryConvert_ULINT_TO_DINT(in, _DINT);
	IF convertResult THEN
		convertAddress := ADR(_DINT);
	END_IF
	
	__SYSTEM.TYPE_CLASS.TYPE_LINT:
	
	convertResult := TryConvert_ULINT_TO_LINT(in, _LINT);
	IF convertResult THEN
		convertAddress := ADR(_LINT);
	END_IF
	
	__SYSTEM.TYPE_CLASS.TYPE_USINT:
	
	convertResult := TryConvert_ULINT_TO_USINT(in, _USINT);
	IF convertResult THEN
		convertAddress := ADR(_USINT);
	END_IF
	
	__SYSTEM.TYPE_CLASS.TYPE_UINT:
	
	convertResult := TryConvert_ULINT_TO_UINT(in, _UINT);
	IF convertResult THEN
		convertAddress := ADR(_UINT);
	END_IF
	
	__SYSTEM.TYPE_CLASS.TYPE_UDINT:
	
	convertResult := TryConvert_ULINT_TO_UDINT(in, _UDINT);
	IF convertResult THEN
		convertAddress := ADR(_UDINT);
	END_IF
	
	__SYSTEM.TYPE_CLASS.TYPE_ULINT:
	
	convertResult := TryConvert_ULINT_TO_ULINT(in, _ULINT);
	IF convertResult THEN
		convertAddress := ADR(_ULINT);
	END_IF
	
	__SYSTEM.TYPE_CLASS.TYPE_REAL:
	
	convertResult := TryConvert_ULINT_TO_REAL(in, _REAL);
	IF convertResult THEN
		convertAddress := ADR(_REAL);
	END_IF
	
	__SYSTEM.TYPE_CLASS.TYPE_LREAL:
	
	convertResult := TryConvert_ULINT_TO_LREAL(in, _LREAL);
	IF convertResult THEN
		convertAddress := ADR(_LREAL);
	END_IF
	
